C05364=1015.142,141.527,-123.022,166.759,55.577,160.204
C05365=1015.138,141.277,-123.003,166.756,55.588,160.206
C05366=1015.133,141.029,-122.984,166.753,55.599,160.207
C05367=1015.129,140.779,-122.966,166.749,55.609,160.208
C05368=1015.125,140.530,-122.946,166.746,55.621,160.210
C05369=1015.120,140.281,-122.928,166.743,55.631,160.211
C05370=1015.116,140.031,-122.909,166.739,55.642,160.212
C05371=1015.111,139.782,-122.890,166.736,55.653,160.214
C05372=1015.107,139.533,-122.872,166.733,55.663,160.215
C05373=1015.102,139.284,-122.852,166.729,55.674,160.217
C05374=1015.097,139.003,-122.832,166.726,55.687,160.218
C05375=1015.092,138.722,-122.810,166.723,55.699,160.220
C05376=1015.087,138.442,-122.789,166.719,55.711,160.221
C05377=1015.083,138.162,-122.768,166.716,55.723,160.223
C05378=1015.079,137.912,-122.749,166.713,55.734,160.225
C05379=1015.074,137.663,-122.731,166.709,55.745,160.226
C05380=1015.070,137.413,-122.712,166.706,55.756,160.228
C05381=1015.065,137.164,-122.694,166.703,55.766,160.229
C05382=1015.061,136.915,-122.674,166.699,55.778,160.230
C05383=1015.056,136.666,-122.656,166.696,55.788,160.232
C05384=1015.052,136.416,-122.637,166.694,55.799,160.233
C05385=1015.047,136.167,-122.619,166.690,55.810,160.235
C05386=1015.043,135.918,-122.600,166.687,55.821,160.236
C05387=1015.039,135.669,-122.582,166.685,55.832,160.238
C05388=1015.035,135.419,-122.563,166.680,55.843,160.239
C05389=1015.030,135.170,-122.545,166.677,55.853,160.240
C05390=1015.025,134.921,-122.527,166.674,55.865,160.242
C05391=1015.021,134.671,-122.508,166.671,55.875,160.243
C05392=1015.016,134.422,-122.489,166.669,55.887,160.245
C05393=1015.012,134.173,-122.470,166.665,55.897,160.246
C05394=1015.008,133.924,-122.453,166.662,55.908,160.247
C05395=1015.003,133.675,-122.434,166.659,55.919,160.249
C05396=1014.999,133.425,-122.416,166.655,55.930,160.250
C05397=1014.994,133.176,-122.397,166.652,55.941,160.252
C05398=1014.990,132.926,-122.379,166.650,55.952,160.253
C05399=1014.985,132.677,-122.361,166.647,55.962,160.255
C05400=1014.981,132.429,-122.342,166.643,55.974,160.256
C05401=1014.977,132.179,-122.323,166.640,55.984,160.258
C05402=1014.972,131.930,-122.305,166.637,55.995,160.259
C05403=1014.967,131.680,-122.287,166.633,56.006,160.260
C05404=1014.963,131.431,-122.268,166.631,56.017,160.262
C05405=1014.959,131.182,-122.250,166.628,56.028,160.263
C05406=1014.955,130.932,-122.232,166.625,56.038,160.265
C05407=1014.950,130.683,-122.214,166.622,56.050,160.266
C05408=1014.945,130.433,-122.195,166.619,56.060,160.268
C05409=1014.942,130.185,-122.177,166.616,56.071,160.269
C05410=1014.937,129.935,-122.159,166.613,56.082,160.271
C05411=1014.933,129.686,-122.140,166.609,56.093,160.272
C05412=1014.928,129.436,-122.122,166.607,56.103,160.273
C05413=1014.924,129.187,-122.104,166.604,56.115,160.275
C05414=1014.919,128.937,-122.086,166.600,56.126,160.276
C05415=1014.915,128.688,-122.068,166.597,56.136,160.278
C05416=1014.910,128.439,-122.050,166.595,56.147,160.279
C05417=1014.905,128.189,-122.032,166.591,56.158,160.281
C05418=1014.901,127.940,-122.014,166.589,56.170,160.282
C05419=1014.896,127.692,-121.996,166.586,56.180,160.284
C05420=1014.892,127.442,-121.979,166.582,56.192,160.285
C05421=1014.887,127.192,-121.961,166.579,56.202,160.287
C05422=1014.882,126.943,-121.942,166.577,56.213,160.288
C05423=1014.878,126.694,-121.925,166.573,56.224,160.290
C05424=1014.873,126.445,-121.906,166.570,56.235,160.291
C05425=1014.869,126.195,-121.889,166.568,56.246,160.293
C05426=1014.865,125.946,-121.871,166.564,56.257,160.294
C05427=1014.860,125.697,-121.853,166.561,56.268,160.295
C05428=1014.856,125.447,-121.835,166.559,56.279,160.297
C05429=1014.851,125.197,-121.817,166.555,56.290,160.298
C05430=1014.847,124.949,-121.799,166.553,56.301,160.300
C05431=1014.842,124.699,-121.781,166.550,56.312,160.301
C05432=1014.838,124.449,-121.763,166.547,56.322,160.303
C05433=1014.834,124.201,-121.746,166.543,56.334,160.304
C05434=1014.829,123.951,-121.728,166.541,56.345,160.306
C05435=1014.825,123.701,-121.710,166.538,56.355,160.307
C05436=1014.820,123.453,-121.692,166.535,56.366,160.309
C05437=1014.816,123.203,-121.674,166.532,56.377,160.310
C05438=1014.810,122.923,-121.654,166.529,56.390,160.312
C05439=1014.805,122.643,-121.634,166.525,56.402,160.314
C05440=1014.800,122.361,-121.615,166.522,56.414,160.315
C05441=1014.796,122.081,-121.594,166.518,56.426,160.317
C05442=1014.791,121.832,-121.576,166.516,56.437,160.318
C05443=1014.787,121.583,-121.558,166.513,56.448,160.320
C05444=1014.782,121.333,-121.541,166.510,56.459,160.321
C05445=1014.777,121.084,-121.523,166.506,56.470,160.322
C05446=1014.773,120.834,-121.506,166.504,56.481,160.324
C05447=1014.769,120.585,-121.488,166.501,56.492,160.326
C05448=1014.764,120.336,-121.469,166.499,56.502,160.327
C05449=1014.760,120.086,-121.452,166.496,56.513,160.328
C05450=1014.755,119.837,-121.434,166.492,56.524,160.330
C05451=1014.751,119.588,-121.417,166.490,56.535,160.331
C05452=1014.747,119.338,-121.399,166.487,56.546,160.333
C05453=1014.742,119.089,-121.381,166.484,56.556,160.334
C05454=1014.738,118.840,-121.364,166.481,56.567,160.336
C05455=1014.733,118.591,-121.346,166.478,56.577,160.337
C05456=1014.729,118.341,-121.328,166.476,56.589,160.339
C05457=1014.725,118.092,-121.310,166.472,56.600,160.340
C05458=1014.721,117.843,-121.293,166.470,56.610,160.342
C05459=1014.716,117.593,-121.275,166.467,56.621,160.343
C05460=1014.711,117.344,-121.257,166.464,56.632,160.344
C05461=1014.707,117.095,-121.240,166.461,56.642,160.346
C05462=1014.702,116.845,-121.222,166.458,56.653,160.347
C05463=1014.699,116.596,-121.205,166.456,56.664,160.349
C05464=1014.694,116.347,-121.186,166.453,56.675,160.350
C05465=1014.690,116.097,-121.169,166.451,56.685,160.352
C05466=1014.685,115.848,-121.151,166.447,56.696,160.353
C05467=1014.681,115.599,-121.134,166.444,56.707,160.355
C05468=1014.676,115.349,-121.116,166.441,56.718,160.356
C05469=1014.672,115.099,-121.098,166.439,56.728,160.357
C05470=1014.668,114.851,-121.081,166.436,56.739,160.359
C05471=1014.663,114.601,-121.063,166.433,56.750,160.360
C05472=1014.659,114.352,-121.045,166.430,56.760,160.362
C05473=1014.655,114.102,-121.028,166.428,56.771,160.363
C05474=1014.651,113.854,-121.010,166.425,56.781,160.365
C05475=1014.646,113.604,-120.993,166.422,56.792,160.366
C05476=1014.642,113.354,-120.976,166.419,56.803,160.368
C05477=1014.637,113.105,-120.957,166.417,56.813,160.369
C05478=1014.634,112.856,-120.940,166.414,56.824,160.370
C05479=1014.629,112.606,-120.922,166.411,56.835,160.372
C05480=1014.625,112.357,-120.905,166.408,56.845,160.373
C05481=1014.620,112.108,-120.887,166.406,56.856,160.375
C05482=1014.616,111.858,-120.870,166.403,56.867,160.376
C05483=1014.612,111.608,-120.852,166.401,56.878,160.378
C05484=1014.608,111.359,-120.835,166.398,56.889,160.379
C05485=1014.602,111.110,-120.818,166.395,56.899,160.381
C05486=1014.598,110.861,-120.801,166.393,56.910,160.382
C05487=1014.595,110.612,-120.784,166.389,56.921,160.384
C05488=1014.590,110.362,-120.766,166.386,56.932,160.385
C05489=1014.585,110.113,-120.749,166.384,56.942,160.387
C05490=1014.581,109.863,-120.732,166.381,56.953,160.388
C05491=1014.577,109.614,-120.715,166.378,56.964,160.389
C05492=1014.572,109.364,-120.698,166.375,56.974,160.391
C05493=1014.568,109.115,-120.681,166.373,56.986,160.393
C05494=1014.563,108.866,-120.662,166.371,56.996,160.394
C05495=1014.558,108.617,-120.646,166.368,57.007,160.396
C05496=1014.554,108.367,-120.628,166.365,57.018,160.397
C05497=1014.549,108.118,-120.612,166.363,57.028,160.398
C05498=1014.545,107.869,-120.595,166.360,57.039,160.400
C05499=1014.540,107.619,-120.578,166.356,57.050,160.401
C05500=1014.536,107.370,-120.561,166.354,57.061,160.403
C05501=1014.531,107.120,-120.544,166.351,57.072,160.404
C05502=1014.526,106.840,-120.526,166.348,57.084,160.406
C05503=1014.521,106.559,-120.505,166.345,57.096,160.408
C05504=1014.516,106.279,-120.486,166.343,57.108,160.409
C05505=1014.511,105.999,-120.468,166.340,57.120,160.411
C05506=1014.507,105.750,-120.451,166.337,57.131,160.412
C05507=1014.502,105.500,-120.434,166.334,57.142,160.414
C05508=1014.498,105.251,-120.417,166.332,57.152,160.415
C05509=1014.493,105.001,-120.400,166.329,57.163,160.417
C05510=1014.489,104.751,-120.383,166.326,57.174,160.418
C05511=1014.485,104.503,-120.366,166.324,57.184,160.420
C05512=1014.480,104.253,-120.349,166.321,57.195,160.421
C05513=1014.476,104.004,-120.332,166.318,57.206,160.423
C05514=1014.471,103.754,-120.315,166.316,57.217,160.424
C05515=1014.467,103.505,-120.298,166.313,57.227,160.426
C05516=1014.463,103.255,-120.281,166.311,57.238,160.427
C05517=1014.458,103.006,-120.265,166.308,57.249,160.429
C05518=1014.454,102.756,-120.247,166.305,57.259,160.430
C05519=1014.449,102.508,-120.231,166.303,57.270,160.432
C05520=1014.445,102.258,-120.214,166.300,57.281,160.433
C05521=1014.440,102.009,-120.197,166.298,57.292,160.435
C05522=1014.436,101.759,-120.180,166.295,57.302,160.436
C05523=1014.431,101.510,-120.163,166.292,57.313,160.437
C05524=1014.427,101.260,-120.146,166.290,57.324,160.439
C05525=1014.422,101.011,-120.130,166.287,57.334,160.440
C05526=1014.418,100.761,-120.113,166.284,57.344,160.442
C05527=1014.414,100.512,-120.096,166.281,57.355,160.443
C05528=1014.410,100.263,-120.079,166.279,57.366,160.445
C05529=1014.405,100.013,-120.062,166.276,57.377,160.446
C05530=1014.401,99.764,-120.045,166.274,57.387,160.448
C05531=1014.396,99.515,-120.029,166.272,57.398,160.449
C05532=1014.392,99.265,-120.012,166.269,57.408,160.450
C05533=1014.387,99.016,-119.995,166.266,57.418,160.452
C05534=1014.383,98.767,-119.978,166.264,57.429,160.453
C05535=1014.379,98.517,-119.962,166.261,57.440,160.455
C05536=1014.374,98.267,-119.945,166.259,57.451,160.456
C05537=1014.369,98.018,-119.929,166.256,57.461,160.458
C05538=1014.365,97.768,-119.912,166.254,57.472,160.459
C05539=1014.361,97.519,-119.896,166.251,57.483,160.461
C05540=1014.356,97.270,-119.879,166.249,57.494,160.462
C05541=1014.351,97.020,-119.863,166.246,57.504,160.464
C05542=1014.347,96.771,-119.846,166.243,57.515,160.465
C05543=1014.342,96.521,-119.829,166.241,57.526,160.467
C05544=1014.338,96.272,-119.814,166.238,57.537,160.468
C05545=1014.333,96.023,-119.797,166.235,57.547,160.469
C05546=1014.329,95.774,-119.781,166.233,57.557,160.471
C05547=1014.324,95.523,-119.764,166.230,57.568,160.472
C05548=1014.320,95.274,-119.747,166.228,57.579,160.474
C05549=1014.315,95.025,-119.731,166.226,57.589,160.476
C05550=1014.311,94.776,-119.715,166.224,57.600,160.477
C05551=1014.306,94.526,-119.698,166.221,57.611,160.479
C05552=1014.302,94.276,-119.682,166.218,57.621,160.480
C05553=1014.298,94.027,-119.665,166.216,57.632,160.481
C05554=1014.293,93.778,-119.649,166.213,57.642,160.483
C05555=1014.289,93.529,-119.633,166.211,57.653,160.484
C05556=1014.283,93.279,-119.616,166.208,57.664,160.486
C05557=1014.280,93.029,-119.600,166.205,57.674,160.487
C05558=1014.275,92.780,-119.583,166.204,57.684,160.489
C05559=1014.271,92.531,-119.567,166.201,57.695,160.490
C05560=1014.266,92.282,-119.551,166.199,57.706,160.492
C05561=1014.261,92.032,-119.534,166.195,57.716,160.493
C05562=1014.258,91.782,-119.518,166.193,57.727,160.494
C05563=1014.253,91.533,-119.501,166.191,57.738,160.496
C05564=1014.249,91.284,-119.486,166.189,57.747,160.497
C05565=1014.244,91.035,-119.469,166.186,57.758,160.499
C05566=1014.239,90.755,-119.451,166.183,57.770,160.500
C05567=1014.234,90.474,-119.432,166.180,57.782,160.502
C05568=1014.228,90.194,-119.414,166.177,57.794,160.504
C05569=1014.224,89.914,-119.395,166.175,57.805,160.506
C05570=1014.219,89.664,-119.379,166.172,57.815,160.507
C05571=1014.215,89.415,-119.363,166.170,57.826,160.508
C05572=1014.211,89.165,-119.346,166.167,57.836,160.509
C05573=1014.207,88.916,-119.330,166.165,57.847,160.511
C05574=1014.202,88.667,-119.314,166.163,57.857,160.513
C05575=1014.197,88.417,-119.298,166.160,57.868,160.514
C05576=1014.193,88.168,-119.282,166.158,57.878,160.515
C05577=1014.189,87.918,-119.266,166.155,57.889,160.517
C05578=1014.184,87.668,-119.250,166.153,57.900,160.518
C05579=1014.180,87.420,-119.234,166.151,57.910,160.520
C05580=1014.175,87.170,-119.218,166.148,57.920,160.521
C05581=1014.170,86.921,-119.203,166.146,57.931,160.523
C05582=1014.165,86.670,-119.187,166.143,57.941,160.524
C05583=1014.161,86.421,-119.170,166.140,57.952,160.526
C05584=1014.156,86.172,-119.154,166.138,57.963,160.527
C05585=1014.152,85.922,-119.138,166.137,57.973,160.529
C05586=1014.148,85.673,-119.122,166.134,57.984,160.530
C05587=1014.143,85.424,-119.106,166.131,57.994,160.532
C05588=1014.139,85.174,-119.090,166.128,58.004,160.533
C05589=1014.134,84.925,-119.075,166.126,58.015,160.534
C05590=1014.129,84.676,-119.059,166.124,58.026,160.536
C05591=1014.125,84.426,-119.043,166.121,58.036,160.537
C05592=1014.120,84.176,-119.027,166.119,58.047,160.539
C05593=1014.116,83.927,-119.011,166.117,58.057,160.540
C05594=1014.111,83.678,-118.995,166.115,58.067,160.542
C05595=1014.107,83.428,-118.979,166.112,58.078,160.543
C05596=1014.103,83.178,-118.963,166.109,58.088,160.545
C05597=1014.098,82.929,-118.947,166.107,58.099,160.546
C05598=1014.093,82.680,-118.932,166.105,58.109,160.547
C05599=1014.089,82.431,-118.916,166.103,58.119,160.549
C05600=1014.084,82.181,-118.900,166.100,58.130,160.550
C05601=1014.080,81.931,-118.884,166.098,58.140,160.552
C05602=1014.076,81.682,-118.868,166.095,58.150,160.553
C05603=1014.071,81.432,-118.853,166.093,58.161,160.555
C05604=1014.067,81.183,-118.836,166.090,58.171,160.556
C05605=1014.062,80.934,-118.820,166.089,58.182,160.558
C05606=1014.057,80.685,-118.805,166.086,58.192,160.559
C05607=1014.053,80.435,-118.789,166.084,58.203,160.560
C05608=1014.049,80.185,-118.774,166.082,58.212,160.562
C05609=1014.044,79.936,-118.758,166.079,58.222,160.563
C05610=1014.040,79.686,-118.742,166.077,58.233,160.565
C05611=1014.036,79.437,-118.726,166.074,58.243,160.566
C05612=1014.031,79.188,-118.710,166.072,58.254,160.568
C05613=1014.027,78.938,-118.694,166.070,58.263,160.569
C05614=1014.022,78.689,-118.679,166.067,58.274,160.570
C05615=1014.018,78.439,-118.663,166.065,58.284,160.572
C05616=1014.013,78.190,-118.647,166.063,58.294,160.573
C05617=1014.009,77.940,-118.632,166.060,58.304,160.575
C05618=1014.005,77.691,-118.616,166.059,58.315,160.576
C05619=1014.000,77.442,-118.599,166.056,58.325,160.578
C05620=1013.996,77.192,-118.584,166.054,58.335,160.579
C05621=1013.991,76.942,-118.568,166.051,58.345,160.580
C05622=1013.986,76.693,-118.553,166.049,58.356,160.582
C05623=1013.982,76.444,-118.537,166.047,58.365,160.583
C05624=1013.978,76.194,-118.521,166.044,58.376,160.584
C05625=1013.973,75.945,-118.506,166.043,58.386,160.586
C05626=1013.968,75.695,-118.490,166.040,58.396,160.587
C05627=1013.964,75.446,-118.474,166.037,58.406,160.589
C05628=1013.959,75.196,-118.460,166.036,58.417,160.590
C05629=1013.955,74.946,-118.444,166.033,58.427,160.592
C05630=1013.950,74.666,-118.426,166.031,58.439,160.594
C05631=1013.945,74.387,-118.409,166.028,58.450,160.595
C05632=1013.940,74.106,-118.392,166.025,58.462,160.597
C05633=1013.935,73.827,-118.374,166.023,58.473,160.598
C05634=1013.930,73.577,-118.360,166.020,58.483,160.599
C05635=1013.926,73.328,-118.344,166.019,58.494,160.601
C05636=1013.921,73.078,-118.329,166.016,58.504,160.602
C05637=1013.917,72.829,-118.313,166.014,58.513,160.604
C05638=1013.912,72.580,-118.298,166.011,58.524,160.605
C05639=1013.907,72.330,-118.282,166.010,58.534,160.607
C05640=1013.903,72.080,-118.266,166.007,58.544,160.608
C05641=1013.898,71.831,-118.252,166.004,58.554,160.609
C05642=1013.894,71.581,-118.236,166.003,58.564,160.611
C05643=1013.889,71.332,-118.221,166.000,58.574,160.612
C05644=1013.885,71.082,-118.205,165.998,58.584,160.614
C05645=1013.880,70.834,-118.190,165.996,58.595,160.615
C05646=1013.876,70.583,-118.175,165.994,58.605,160.617
C05647=1013.872,70.334,-118.160,165.991,58.615,160.618
C05648=1013.867,70.085,-118.144,165.989,58.625,160.619
C05649=1013.863,69.835,-118.129,165.986,58.635,160.621
C05650=1013.857,69.586,-118.114,165.985,58.645,160.622
C05651=1013.853,69.335,-118.098,165.982,58.655,160.623
C05652=1013.848,69.086,-118.083,165.981,58.665,160.625
C05653=1013.845,68.837,-118.068,165.978,58.676,160.626
C05654=1013.840,68.588,-118.053,165.976,58.685,160.628
C05655=1013.836,68.338,-118.038,165.974,58.695,160.629
C05656=1013.831,68.088,-118.022,165.971,58.705,160.631
C05657=1013.826,67.839,-118.007,165.970,58.715,160.632
C05658=1013.822,67.589,-117.992,165.967,58.725,160.633
C05659=1013.817,67.340,-117.977,165.965,58.735,160.635
C05660=1013.813,67.091,-117.962,165.962,58.745,160.636
C05661=1013.809,66.841,-117.947,165.960,58.755,160.637
C05662=1013.804,66.592,-117.931,165.958,58.765,160.639
C05663=1013.799,66.342,-117.917,165.956,58.775,160.640
C05664=1013.795,66.092,-117.901,165.953,58.785,160.641
C05665=1013.790,65.843,-117.886,165.951,58.795,160.643
C05666=1013.786,65.593,-117.871,165.950,58.805,160.644
C05667=1013.781,65.344,-117.856,165.947,58.815,160.646
C05668=1013.777,65.094,-117.842,165.945,58.825,160.647
C05669=1013.772,64.845,-117.826,165.942,58.835,160.648
C05670=1013.767,64.595,-117.811,165.940,58.845,160.650
C05671=1013.762,64.345,-117.796,165.939,58.855,160.651
C05672=1013.759,64.097,-117.781,165.936,58.865,160.653
C05673=1013.754,63.847,-117.766,165.934,58.875,160.654
C05674=1013.749,63.597,-117.751,165.931,58.885,160.655
C05675=1013.745,63.347,-117.736,165.930,58.895,160.657
C05676=1013.741,63.099,-117.721,165.928,58.904,160.658
C05677=1013.736,62.849,-117.707,165.925,58.915,160.660
C05678=1013.731,62.599,-117.691,165.924,58.924,160.661
C05679=1013.727,62.349,-117.677,165.922,58.934,160.663
C05680=1013.722,62.099,-117.662,165.919,58.944,160.664
C05681=1013.718,61.851,-117.647,165.917,58.954,160.665
C05682=1013.713,61.601,-117.633,165.915,58.964,160.667
C05683=1013.708,61.351,-117.619,165.913,58.974,160.668
C05684=1013.703,61.102,-117.603,165.910,58.984,160.669
C05685=1013.699,60.853,-117.589,165.908,58.994,160.671
C05686=1013.694,60.603,-117.575,165.906,59.005,160.672
C05687=1013.689,60.353,-117.560,165.904,59.014,160.674
C05688=1013.684,60.104,-117.545,165.902,59.024,160.675
C05689=1013.680,59.854,-117.531,165.899,59.034,160.676
C05690=1013.675,59.605,-117.516,165.897,59.043,160.678
C05691=1013.670,59.355,-117.501,165.894,59.054,160.679
C05692=1013.666,59.105,-117.487,165.893,59.064,160.680
C05693=1013.662,58.856,-117.473,165.891,59.073,160.682
C05694=1013.656,58.576,-117.456,165.888,59.085,160.683
C05695=1013.651,58.296,-117.439,165.886,59.096,160.685
C05696=1013.646,58.016,-117.424,165.884,59.107,160.687
C05697=1013.641,57.737,-117.407,165.882,59.118,160.688
C05698=1013.636,57.487,-117.393,165.878,59.127,160.689
C05699=1013.631,57.238,-117.378,165.877,59.137,160.691
C05700=1013.626,56.988,-117.363,165.875,59.147,160.692
C05701=1013.622,56.739,-117.349,165.873,59.157,160.694
C05702=1013.617,56.489,-117.335,165.870,59.166,160.695
C05703=1013.613,56.239,-117.320,165.868,59.176,160.696
C05704=1013.608,55.990,-117.306,165.867,59.186,160.698
C05705=1013.604,55.741,-117.291,165.865,59.196,160.699
C05706=1013.599,55.491,-117.277,165.862,59.205,160.700
C05707=1013.595,55.241,-117.263,165.860,59.215,160.702
C05708=1013.590,54.992,-117.248,165.859,59.225,160.703
C05709=1013.585,54.742,-117.233,165.856,59.234,160.704
C05710=1013.581,54.493,-117.219,165.854,59.244,160.705
C05711=1013.576,54.243,-117.204,165.851,59.253,160.707
C05712=1013.571,53.993,-117.190,165.850,59.263,160.708
C05713=1013.567,53.744,-117.176,165.848,59.273,160.710
C05714=1013.562,53.495,-117.161,165.846,59.282,160.711
C05715=1013.557,53.245,-117.146,165.843,59.293,160.712
C05716=1013.553,52.996,-117.132,165.841,59.302,160.713
C05717=1013.549,52.746,-117.118,165.839,59.311,160.715
C05718=1013.544,52.497,-117.103,165.837,59.321,160.716
C05719=1013.540,52.247,-117.089,165.835,59.330,160.718
C05720=1013.535,51.997,-117.075,165.833,59.340,160.719
C05721=1013.530,51.748,-117.060,165.832,59.349,160.720
C05722=1013.526,51.499,-117.045,165.829,59.358,160.721
C05723=1013.521,51.249,-117.031,165.827,59.369,160.723
C05724=1013.517,50.999,-117.017,165.824,59.378,160.724
C05725=1013.513,50.749,-117.002,165.822,59.387,160.725
C05726=1013.509,50.500,-116.988,165.821,59.397,160.727
C05727=1013.504,50.250,-116.973,165.818,59.406,160.728
C05728=1013.499,50.000,-116.959,165.817,59.416,160.729
C05729=1013.495,49.751,-116.945,165.814,59.425,160.731
C05730=1013.490,49.502,-116.929,165.812,59.434,160.732
C05731=1013.486,49.253,-116.915,165.811,59.444,160.733
C05732=1013.481,49.003,-116.901,165.808,59.453,160.734
C05733=1013.477,48.754,-116.887,165.806,59.462,160.736
C05734=1013.472,48.504,-116.872,165.804,59.471,160.737
C05735=1013.468,48.254,-116.858,165.802,59.481,160.738
C05736=1013.463,48.005,-116.844,165.800,59.490,160.740
C05737=1013.459,47.755,-116.829,165.798,59.499,160.741
C05738=1013.455,47.506,-116.815,165.796,59.509,160.742
C05739=1013.450,47.256,-116.801,165.794,59.518,160.743
C05740=1013.446,47.007,-116.787,165.792,59.528,160.745
C05741=1013.441,46.757,-116.772,165.790,59.537,160.746
C05742=1013.436,46.507,-116.758,165.788,59.546,160.747
C05743=1013.432,46.258,-116.744,165.785,59.555,160.748
C05744=1013.427,46.008,-116.729,165.784,59.564,160.750
C05745=1013.423,45.758,-116.715,165.783,59.573,160.751
C05746=1013.418,45.509,-116.701,165.781,59.583,160.752
C05747=1013.414,45.259,-116.687,165.778,59.592,160.754
C05748=1013.410,45.010,-116.672,165.776,59.601,160.755
C05749=1013.405,44.760,-116.658,165.774,59.610,160.756
C05750=1013.401,44.510,-116.644,165.772,59.619,160.757
C05751=1013.397,44.261,-116.629,165.770,59.628,160.758
C05752=1013.392,44.011,-116.615,165.768,59.637,160.760
C05753=1013.388,43.762,-116.601,165.766,59.646,160.761
C05754=1013.383,43.512,-116.586,165.764,59.655,160.762
C05755=1013.379,43.263,-116.572,165.762,59.664,160.763
C05756=1013.374,43.013,-116.558,165.760,59.674,160.765
C05757=1013.370,42.764,-116.544,165.759,59.682,160.766
C05758=1013.365,42.485,-116.527,165.756,59.693,160.767
C05759=1013.360,42.205,-116.512,165.754,59.703,160.769
C05760=1013.355,41.925,-116.496,165.751,59.712,160.770
C05761=1013.350,41.645,-116.481,165.749,59.722,160.771
C05762=1013.345,41.395,-116.466,165.747,59.732,160.772
C05763=1013.340,41.146,-116.453,165.744,59.741,160.774
C05764=1013.335,40.896,-116.438,165.743,59.749,160.775
C05765=1013.332,40.646,-116.425,165.741,59.759,160.776
C05766=1013.327,40.396,-116.410,165.739,59.768,160.777
C05767=1013.322,40.147,-116.397,165.737,59.777,160.779
C05768=1013.318,39.898,-116.383,165.735,59.786,160.780
C05769=1013.313,39.648,-116.369,165.734,59.795,160.781
C05770=1013.308,39.399,-116.356,165.732,59.804,160.782
C05771=1013.304,39.149,-116.341,165.729,59.813,160.784
C05772=1013.300,38.900,-116.327,165.727,59.822,160.785
C05773=1013.295,38.649,-116.313,165.726,59.831,160.786
C05774=1013.290,38.400,-116.300,165.724,59.840,160.788
C05775=1013.286,38.151,-116.285,165.721,59.849,160.788
C05776=1013.282,37.901,-116.272,165.719,59.858,160.790
C05777=1013.277,37.652,-116.258,165.718,59.867,160.791
C05778=1013.272,37.402,-116.244,165.716,59.876,160.792
C05779=1013.268,37.153,-116.230,165.713,59.884,160.793
C05780=1013.263,36.903,-116.217,165.712,59.893,160.795
C05781=1013.259,36.653,-116.203,165.710,59.902,160.796
C05782=1013.255,36.404,-116.189,165.708,59.911,160.797
C05783=1013.250,36.154,-116.175,165.706,59.919,160.798
C05784=1013.245,35.905,-116.161,165.704,59.928,160.799
C05785=1013.241,35.654,-116.148,165.702,59.938,160.801
C05786=1013.236,35.406,-116.134,165.700,59.947,160.802
C05787=1013.231,35.156,-116.121,165.698,59.955,160.803
C05788=1013.227,34.906,-116.107,165.696,59.964,160.804
C05789=1013.222,34.657,-116.094,165.694,59.973,160.805
C05790=1013.217,34.407,-116.080,165.693,59.982,160.807
C05791=1013.213,34.157,-116.067,165.690,59.990,160.808
C05792=1013.209,33.908,-116.053,165.688,59.999,160.809
C05793=1013.203,33.658,-116.040,165.687,60.008,160.810
C05794=1013.199,33.409,-116.025,165.684,60.017,160.811
C05795=1013.195,33.159,-116.013,165.682,60.026,160.812
C05796=1013.189,32.910,-115.999,165.681,60.035,160.814
C05797=1013.185,32.660,-115.985,165.678,60.043,160.815
C05798=1013.181,32.411,-115.972,165.676,60.052,160.816
C05799=1013.176,32.160,-115.958,165.674,60.060,160.817
C05800=1013.172,31.911,-115.945,165.672,60.069,160.818
C05801=1013.167,31.662,-115.931,165.671,60.078,160.820
C05802=1013.162,31.412,-115.918,165.669,60.087,160.821
C05803=1013.158,31.162,-115.904,165.668,60.095,160.822
C05804=1013.154,30.913,-115.891,165.665,60.104,160.823
C05805=1013.148,30.663,-115.877,165.663,60.112,160.824
C05806=1013.144,30.414,-115.864,165.661,60.121,160.825
C05807=1013.140,30.164,-115.851,165.659,60.129,160.826
C05808=1013.135,29.914,-115.837,165.657,60.138,160.828
C05809=1013.130,29.665,-115.824,165.656,60.146,160.829
C05810=1013.126,29.415,-115.810,165.654,60.155,160.830
C05811=1013.121,29.165,-115.797,165.652,60.163,160.831
C05812=1013.117,28.915,-115.783,165.649,60.172,160.832
C05813=1013.112,28.667,-115.770,165.648,60.181,160.833
C05814=1013.107,28.416,-115.757,165.646,60.189,160.834
C05815=1013.103,28.167,-115.743,165.644,60.197,160.835
C05816=1013.098,27.918,-115.730,165.642,60.206,160.837
C05817=1013.095,27.668,-115.717,165.640,60.214,160.838
C05818=1013.089,27.418,-115.703,165.638,60.222,160.839
C05819=1013.085,27.169,-115.689,165.636,60.231,160.840
C05820=1013.081,26.919,-115.677,165.635,60.240,160.841
C05821=1013.076,26.669,-115.663,165.632,60.248,160.842
C05822=1013.071,26.430,-115.650,165.630,60.256,160.843
C05823=1013.067,26.191,-115.638,165.629,60.264,160.844
C05824=1013.063,25.951,-115.625,165.627,60.272,160.845
C05825=1013.058,25.712,-115.612,165.625,60.280,160.847
C05826=1013.054,25.474,-115.600,165.624,60.288,160.848
C05827=1013.049,25.234,-115.587,165.622,60.296,160.849
C05828=1013.045,24.994,-115.575,165.620,60.303,160.850
C05829=1013.041,24.756,-115.562,165.617,60.312,160.850
C05830=1013.036,24.506,-115.549,165.616,60.321,160.852
C05831=1013.031,24.256,-115.536,165.615,60.329,160.853
C05832=1013.026,24.006,-115.523,165.612,60.337,160.854
C05833=1013.022,23.757,-115.510,165.610,60.345,160.855
C05834=1013.018,23.507,-115.497,165.609,60.353,160.856
C05835=1013.014,23.258,-115.484,165.606,60.362,160.857
C05836=1013.008,23.008,-115.470,165.604,60.370,160.858
C05837=1013.003,22.758,-115.457,165.603,60.378,160.859
C05838=1012.999,22.509,-115.444,165.601,60.386,160.860
C05839=1012.995,22.259,-115.431,165.598,60.394,160.861
C05840=1012.990,22.010,-115.418,165.597,60.402,160.862
C05841=1012.985,21.759,-115.405,165.595,60.410,160.864
C05842=1012.981,21.510,-115.392,165.593,60.418,160.865
C05843=1012.976,21.260,-115.380,165.591,60.427,160.866
C05844=1012.972,21.011,-115.365,165.589,60.435,160.867
C05845=1012.967,20.762,-115.353,165.588,60.443,160.868
C05846=1012.962,20.512,-115.340,165.586,60.451,160.869
C05847=1012.958,20.262,-115.327,165.584,60.459,160.870
C05848=1012.953,20.013,-115.314,165.582,60.468,160.871
C05849=1012.949,19.763,-115.301,165.580,60.476,160.872
C05850=1012.945,19.513,-115.288,165.578,60.484,160.873
C05851=1012.940,19.264,-115.275,165.576,60.491,160.874
C05852=1012.935,19.014,-115.262,165.575,60.499,160.875
C05853=1012.930,18.764,-115.249,165.573,60.507,160.876
C05854=1012.926,18.515,-115.236,165.571,60.515,160.877
C05855=1012.921,18.265,-115.224,165.570,60.523,160.878
C05856=1012.917,18.016,-115.211,165.566,60.531,160.879
C05857=1012.912,17.766,-115.198,165.565,60.539,160.880
C05858=1012.908,17.517,-115.185,165.563,60.547,160.881
C05859=1012.903,17.266,-115.171,165.562,60.555,160.882
C05860=1012.899,17.017,-115.159,165.559,60.562,160.883
C05861=1012.894,16.767,-115.146,165.558,60.570,160.884
C05862=1012.889,16.518,-115.133,165.556,60.578,160.885
C05863=1012.885,16.268,-115.120,165.554,60.586,160.886
C05864=1012.880,16.019,-115.108,165.552,60.594,160.887
C05865=1012.876,15.769,-115.095,165.551,60.602,160.888
C05866=1012.872,15.519,-115.083,165.548,60.609,160.889
C05867=1012.867,15.270,-115.070,165.547,60.617,160.890
C05868=1012.862,15.019,-115.057,165.545,60.625,160.891
C05869=1012.857,14.770,-115.044,165.543,60.632,160.892
C05870=1012.853,14.520,-115.031,165.541,60.641,160.893
C05871=1012.848,14.271,-115.018,165.539,60.648,160.894
C05872=1012.844,14.021,-115.006,165.538,60.656,160.895
C05873=1012.839,13.772,-114.993,165.535,60.663,160.896
C05874=1012.835,13.522,-114.981,165.534,60.671,160.897
C05875=1012.830,13.272,-114.968,165.532,60.679,160.898
C05876=1012.826,13.023,-114.955,165.530,60.687,160.899
C05877=1012.821,12.773,-114.942,165.528,60.694,160.900
C05878=1012.809,24.482,-115.964,165.590,60.551,160.891
C05879=1012.813,24.732,-115.977,165.592,60.543,160.889
C05880=1012.818,24.982,-115.990,165.593,60.535,160.888
C05881=1012.823,25.231,-116.003,165.595,60.527,160.887
C05882=1012.827,25.481,-116.016,165.596,60.519,160.886
C05883=1012.832,25.770,-116.031,165.599,60.509,160.885
C05884=1012.838,26.059,-116.047,165.601,60.500,160.884
C05885=1012.843,26.347,-116.061,165.603,60.490,160.883
C05886=1012.848,26.637,-116.077,165.605,60.481,160.881
C05887=1012.853,26.887,-116.090,165.607,60.473,160.880
C05888=1012.858,27.136,-116.103,165.610,60.465,160.879
C05889=1012.862,27.385,-116.117,165.611,60.457,160.878
C05890=1012.867,27.635,-116.130,165.613,60.449,160.877
C05891=1012.871,27.885,-116.143,165.615,60.441,160.876
C05892=1012.875,28.135,-116.156,165.616,60.433,160.875
C05893=1012.879,28.384,-116.170,165.619,60.424,160.874
C05894=1012.885,28.634,-116.183,165.620,60.416,160.873
C05895=1012.888,28.884,-116.197,165.622,60.408,160.872
C05896=1012.893,29.133,-116.210,165.624,60.400,160.870
C05897=1012.898,29.382,-116.223,165.626,60.391,160.870
C05898=1012.902,29.633,-116.237,165.628,60.383,160.868
C05899=1012.907,29.882,-116.250,165.629,60.375,160.867
C05900=1012.911,30.131,-116.264,165.630,60.367,160.866
C05901=1012.916,30.381,-116.276,165.633,60.358,160.865
C05902=1012.920,30.631,-116.291,165.635,60.350,160.864
C05903=1012.925,30.880,-116.304,165.636,60.342,160.863
C05904=1012.929,31.129,-116.318,165.639,60.334,160.862
C05905=1012.934,31.380,-116.331,165.640,60.325,160.860
C05906=1012.939,31.629,-116.344,165.643,60.316,160.859
C05907=1012.943,31.878,-116.358,165.644,60.308,160.858
C05908=1012.947,32.128,-116.371,165.645,60.300,160.857
C05909=1012.952,32.378,-116.385,165.648,60.291,160.856
C05910=1012.957,32.627,-116.398,165.650,60.283,160.855
C05911=1012.961,32.877,-116.411,165.652,60.275,160.854
C05912=1012.966,33.127,-116.425,165.653,60.266,160.852
C05913=1012.970,33.376,-116.438,165.655,60.258,160.851
C05914=1012.975,33.625,-116.452,165.657,60.249,160.850
C05915=1012.980,33.875,-116.465,165.659,60.241,160.849
C05916=1012.984,34.125,-116.478,165.661,60.232,160.848
C05917=1012.989,34.374,-116.492,165.662,60.223,160.847
C05918=1012.992,34.624,-116.505,165.665,60.215,160.846
C05919=1012.998,34.874,-116.519,165.666,60.206,160.844
C05920=1013.002,35.123,-116.533,165.669,60.198,160.843
C05921=1013.007,35.372,-116.546,165.671,60.188,160.842
C05922=1013.011,35.623,-116.560,165.673,60.180,160.841
C05923=1013.016,35.872,-116.573,165.675,60.171,160.840
C05924=1013.020,36.122,-116.587,165.676,60.163,160.839
C05925=1013.025,36.371,-116.600,165.678,60.154,160.837
C05926=1013.029,36.621,-116.614,165.680,60.146,160.836
C05927=1013.034,36.871,-116.628,165.682,60.137,160.835
C05928=1013.038,37.120,-116.641,165.684,60.129,160.834
C05929=1013.043,37.369,-116.655,165.686,60.120,160.833
C05930=1013.047,37.619,-116.670,165.687,60.112,160.832
C05931=1013.052,37.869,-116.682,165.689,60.102,160.830
C05932=1013.057,38.119,-116.697,165.690,60.094,160.829
C05933=1013.060,38.368,-116.710,165.693,60.085,160.828
C05934=1013.065,38.618,-116.724,165.695,60.076,160.827
C05935=1013.070,38.867,-116.738,165.697,60.068,160.826
C05936=1013.074,39.117,-116.752,165.699,60.059,160.824
C05937=1013.078,39.366,-116.766,165.700,60.050,160.823
C05938=1013.083,39.616,-116.780,165.703,60.042,160.822
C05939=1013.087,39.866,-116.793,165.705,60.032,160.821
C05940=1013.092,40.115,-116.807,165.706,60.024,160.819
C05941=1013.096,40.365,-116.822,165.709,60.015,160.819
C05942=1013.101,40.613,-116.835,165.711,60.006,160.817
C05943=1013.105,40.864,-116.849,165.712,59.997,160.816
C05944=1013.110,41.113,-116.863,165.714,59.988,160.815
C05945=1013.115,41.363,-116.877,165.717,59.980,160.814
C05946=1013.119,41.613,-116.890,165.719,59.971,160.813
C05947=1013.124,41.892,-116.906,165.720,59.961,160.811
C05948=1013.129,42.172,-116.922,165.722,59.951,160.809
C05949=1013.134,42.452,-116.938,165.725,59.941,160.808
C05950=1013.139,42.731,-116.954,165.726,59.931,160.807
C05951=1013.144,42.980,-116.968,165.728,59.922,160.806
C05952=1013.147,43.230,-116.981,165.731,59.914,160.805
C05953=1013.152,43.480,-116.996,165.732,59.905,160.803
C05954=1013.156,43.729,-117.010,165.734,59.896,160.802
C05955=1013.161,43.979,-117.024,165.736,59.886,160.801
C05956=1013.165,44.228,-117.038,165.737,59.878,160.799
C05957=1013.170,44.478,-117.053,165.740,59.869,160.798
C05958=1013.174,44.728,-117.067,165.742,59.860,160.797
C05959=1013.178,44.977,-117.081,165.745,59.851,160.796
C05960=1013.183,45.227,-117.096,165.746,59.842,160.795
C05961=1013.187,45.476,-117.110,165.748,59.833,160.793
C05962=1013.192,45.726,-117.124,165.750,59.824,160.792
C05963=1013.196,45.975,-117.138,165.752,59.815,160.791
C05964=1013.201,46.225,-117.153,165.753,59.806,160.789
C05965=1013.205,46.474,-117.167,165.755,59.797,160.788
C05966=1013.210,46.724,-117.181,165.757,59.788,160.787
C05967=1013.214,46.973,-117.195,165.759,59.779,160.786
C05968=1013.218,47.223,-117.210,165.762,59.769,160.785
C05969=1013.223,47.472,-117.224,165.763,59.761,160.783
C05970=1013.227,47.722,-117.238,165.765,59.752,160.782
C05971=1013.231,47.971,-117.252,165.767,59.742,160.781
C05972=1013.236,48.221,-117.267,165.769,59.733,160.780
C05973=1013.240,48.470,-117.281,165.771,59.724,160.778
C05974=1013.245,48.720,-117.295,165.773,59.715,160.777
C05975=1013.249,48.969,-117.310,165.776,59.706,160.776
C05976=1013.254,49.219,-117.324,165.778,59.697,160.775
C05977=1013.259,49.469,-117.338,165.780,59.687,160.774
C05978=1013.263,49.718,-117.353,165.781,59.679,160.772
C05979=1013.268,49.968,-117.367,165.783,59.669,160.771
C05980=1013.272,50.217,-117.381,165.785,59.660,160.769
C05981=1013.276,50.467,-117.396,165.787,59.651,160.768
C05982=1013.281,50.716,-117.410,165.789,59.641,160.767
C05983=1013.285,50.966,-117.424,165.791,59.632,160.766
C05984=1013.289,51.215,-117.438,165.793,59.622,160.764
C05985=1013.294,51.465,-117.453,165.795,59.613,160.763
C05986=1013.298,51.714,-117.467,165.797,59.604,160.762
C05987=1013.303,51.964,-117.481,165.799,59.594,160.760
C05988=1013.308,52.214,-117.496,165.801,59.585,160.759
C05989=1013.312,52.463,-117.510,165.803,59.576,160.758
C05990=1013.317,52.713,-117.524,165.805,59.566,160.756
C05991=1013.321,52.963,-117.538,165.807,59.557,160.755
C05992=1013.326,53.212,-117.553,165.809,59.548,160.754
C05993=1013.330,53.462,-117.567,165.810,59.538,160.752
C05994=1013.335,53.711,-117.582,165.814,59.528,160.751
C05995=1013.339,53.961,-117.597,165.816,59.519,160.750
C05996=1013.343,54.210,-117.611,165.818,59.509,160.749
C05997=1013.348,54.460,-117.626,165.820,59.500,160.747
C05998=1013.352,54.710,-117.640,165.821,59.490,160.746
C05999=1013.356,54.959,-117.654,165.824,59.481,160.745
C06000=1013.361,55.209,-117.669,165.825,59.471,160.743
C06001=1013.365,55.458,-117.683,165.827,59.462,160.742
C06002=1013.370,55.708,-117.698,165.830,59.452,160.741
C06003=1013.375,55.957,-117.712,165.832,59.443,160.739
C06004=1013.379,56.207,-117.726,165.834,59.433,160.738
C06005=1013.384,56.457,-117.741,165.836,59.424,160.737
C06006=1013.388,56.706,-117.755,165.837,59.414,160.735
C06007=1013.393,56.956,-117.769,165.839,59.404,160.734
C06008=1013.398,57.205,-117.784,165.842,59.395,160.733
C06009=1013.402,57.454,-117.799,165.844,59.385,160.731
C06010=1013.407,57.704,-117.813,165.846,59.376,160.730
C06011=1013.412,57.983,-117.830,165.848,59.365,160.728
C06012=1013.417,58.263,-117.845,165.850,59.354,160.727
C06013=1013.422,58.543,-117.861,165.853,59.342,160.725
C06014=1013.428,58.822,-117.878,165.856,59.332,160.724
C06015=1013.432,59.072,-117.892,165.858,59.322,160.722
C06016=1013.437,59.322,-117.907,165.859,59.312,160.721
C06017=1013.441,59.571,-117.921,165.862,59.302,160.720
C06018=1013.446,59.821,-117.935,165.864,59.293,160.718
C06019=1013.451,60.070,-117.950,165.866,59.283,160.717
C06020=1013.455,60.319,-117.964,165.868,59.273,160.716
C06021=1013.460,60.569,-117.979,165.870,59.263,160.714
C06022=1013.464,60.819,-117.994,165.872,59.253,160.713
C06023=1013.469,61.069,-118.009,165.875,59.243,160.712
C06024=1013.473,61.318,-118.023,165.877,59.234,160.710
C06025=1013.478,61.568,-118.038,165.878,59.224,160.709
C06026=1013.483,61.818,-118.052,165.881,59.213,160.707
C06027=1013.487,62.066,-118.067,165.882,59.204,160.706
C06028=1013.492,62.316,-118.081,165.884,59.194,160.704
C06029=1013.496,62.566,-118.096,165.887,59.183,160.703
C06030=1013.502,62.815,-118.111,165.889,59.174,160.702
C06031=1013.505,63.065,-118.126,165.891,59.165,160.700
C06032=1013.510,63.315,-118.140,165.893,59.154,160.699
C06033=1013.515,63.564,-118.155,165.895,59.144,160.698
C06034=1013.519,63.814,-118.170,165.897,59.135,160.696
C06035=1013.523,64.063,-118.185,165.900,59.125,160.695
C06036=1013.528,64.313,-118.200,165.902,59.115,160.694
C06037=1013.532,64.562,-118.216,165.903,59.106,160.692
C06038=1013.537,64.812,-118.230,165.906,59.095,160.691
C06039=1013.541,65.061,-118.245,165.908,59.085,160.689
C06040=1013.545,65.311,-118.260,165.909,59.076,160.688
C06041=1013.550,65.560,-118.275,165.912,59.065,160.686
C06042=1013.555,65.810,-118.289,165.914,59.056,160.685
C06043=1013.559,66.059,-118.305,165.917,59.046,160.684
C06044=1013.564,66.309,-118.319,165.919,59.036,160.683
C06045=1013.568,66.558,-118.335,165.921,59.026,160.681
C06046=1013.573,66.808,-118.350,165.923,59.016,160.680
C06047=1013.578,67.057,-118.365,165.925,59.006,160.678
C06048=1013.581,67.306,-118.380,165.928,58.996,160.677
C06049=1013.586,67.556,-118.395,165.929,58.986,160.675
C06050=1013.590,67.806,-118.410,165.931,58.977,160.674
C06051=1013.595,68.056,-118.425,165.934,58.966,160.673
C06052=1013.599,68.305,-118.441,165.936,58.956,160.671
C06053=1013.604,68.554,-118.455,165.938,58.946,160.670
C06054=1013.608,68.804,-118.470,165.940,58.936,160.668
C06055=1013.613,69.053,-118.486,165.942,58.927,160.667
C06056=1013.617,69.303,-118.501,165.945,58.916,160.666
C06057=1013.622,69.553,-118.516,165.946,58.907,160.664
C06058=1013.626,69.802,-118.531,165.949,58.896,160.663
C06059=1013.631,70.051,-118.546,165.951,58.887,160.661
C06060=1013.635,70.301,-118.561,165.954,58.876,160.660
C06061=1013.640,70.550,-118.577,165.955,58.867,160.659
C06062=1013.644,70.800,-118.592,165.958,58.856,160.657
C06063=1013.648,71.049,-118.608,165.960,58.847,160.656
C06064=1013.653,71.299,-118.622,165.963,58.836,160.655
C06065=1013.657,71.548,-118.638,165.964,58.827,160.653
C06066=1013.662,71.798,-118.653,165.967,58.816,160.652
C06067=1013.666,72.047,-118.669,165.968,58.806,160.650
C06068=1013.670,72.297,-118.684,165.971,58.796,160.649
C06069=1013.675,72.547,-118.699,165.973,58.786,160.647
C06070=1013.680,72.796,-118.715,165.976,58.776,160.646
C06071=1013.684,73.045,-118.730,165.977,58.766,160.645
C06072=1013.688,73.294,-118.746,165.980,58.756,160.643
C06073=1013.693,73.544,-118.760,165.981,58.745,160.641
C06074=1013.697,73.794,-118.776,165.984,58.735,160.640
C06075=1013.702,74.073,-118.793,165.986,58.724,160.639
C06076=1013.707,74.353,-118.811,165.989,58.713,160.637
C06077=1013.712,74.633,-118.828,165.991,58.701,160.635
C06078=1013.718,74.913,-118.844,165.994,58.690,160.634
C06079=1013.722,75.163,-118.860,165.995,58.679,160.632
C06080=1013.726,75.412,-118.876,165.998,58.669,160.631
C06081=1013.731,75.661,-118.891,166.001,58.659,160.630
C06082=1013.735,75.910,-118.906,166.003,58.649,160.628
C06083=1013.739,76.160,-118.922,166.005,58.638,160.627
C06084=1013.745,76.409,-118.937,166.007,58.628,160.625
C06085=1013.749,76.659,-118.953,166.010,58.618,160.624
C06086=1013.753,76.909,-118.968,166.013,58.608,160.623
C06087=1013.757,77.158,-118.984,166.014,58.597,160.621
C06088=1013.762,77.408,-118.999,166.017,58.587,160.620
C06089=1013.767,77.657,-119.016,166.018,58.577,160.618
C06090=1013.771,77.906,-119.031,166.021,58.567,160.617
C06091=1013.775,78.156,-119.047,166.022,58.557,160.615
C06092=1013.780,78.405,-119.063,166.025,58.547,160.614
C06093=1013.784,78.655,-119.079,166.028,58.536,160.613
C06094=1013.788,78.905,-119.094,166.030,58.527,160.611
C06095=1013.792,79.153,-119.110,166.032,58.516,160.610
C06096=1013.797,79.403,-119.125,166.034,58.506,160.608
C06097=1013.801,79.652,-119.141,166.037,58.496,160.607
C06098=1013.806,79.902,-119.157,166.039,58.485,160.605
C06099=1013.810,80.151,-119.172,166.041,58.475,160.604
C06100=1013.814,80.401,-119.188,166.044,58.465,160.603
C06101=1013.819,80.651,-119.204,166.046,58.454,160.601
C06102=1013.823,80.900,-119.220,166.048,58.444,160.600
C06103=1013.827,81.150,-119.235,166.050,58.434,160.598
C06104=1013.832,81.399,-119.252,166.053,58.423,160.597
C06105=1013.837,81.648,-119.267,166.055,58.414,160.595
C06106=1013.841,81.898,-119.283,166.057,58.403,160.594
C06107=1013.845,82.147,-119.299,166.060,58.393,160.592
C06108=1013.850,82.397,-119.314,166.061,58.382,160.591
C06109=1013.854,82.646,-119.330,166.064,58.372,160.589
C06110=1013.858,82.896,-119.346,166.067,58.361,160.588
C06111=1013.863,83.145,-119.362,166.070,58.351,160.587
C06112=1013.867,83.394,-119.378,166.071,58.341,160.585
C06113=1013.872,83.644,-119.393,166.074,58.330,160.584
C06114=1013.877,83.893,-119.409,166.076,58.320,160.582
C06115=1013.881,84.143,-119.425,166.079,58.309,160.581
C06116=1013.885,84.392,-119.441,166.080,58.299,160.579
C06117=1013.890,84.642,-119.456,166.083,58.289,160.578
C06118=1013.894,84.892,-119.472,166.085,58.278,160.576
C06119=1013.898,85.141,-119.489,166.088,58.267,160.575
C06120=1013.903,85.390,-119.504,166.090,58.257,160.573
C06121=1013.908,85.639,-119.520,166.092,58.246,160.572
C06122=1013.912,85.889,-119.535,166.095,58.236,160.571
C06123=1013.916,86.139,-119.551,166.097,58.225,160.569
C06124=1013.922,86.388,-119.568,166.100,58.215,160.567
C06125=1013.926,86.638,-119.584,166.102,58.204,160.566
C06126=1013.930,86.887,-119.600,166.104,58.194,160.564
C06127=1013.935,87.137,-119.615,166.106,58.183,160.563
C06128=1013.939,87.386,-119.632,166.109,58.173,160.562
C06129=1013.943,87.635,-119.648,166.111,58.162,160.560
C06130=1013.949,87.885,-119.663,166.114,58.151,160.559
C06131=1013.953,88.134,-119.679,166.117,58.141,160.557
C06132=1013.957,88.384,-119.694,166.119,58.130,160.556
C06133=1013.962,88.633,-119.711,166.120,58.120,160.554
C06134=1013.966,88.882,-119.727,166.123,58.110,160.553
C06135=1013.970,89.132,-119.744,166.126,58.099,160.551
C06136=1013.975,89.382,-119.760,166.128,58.088,160.550
C06137=1013.979,89.632,-119.776,166.131,58.078,160.549
C06138=1013.984,89.880,-119.792,166.132,58.068,160.547
C06139=1013.988,90.161,-119.811,166.135,58.056,160.545
C06140=1013.994,90.440,-119.829,166.139,58.044,160.544
C06141=1013.998,90.720,-119.846,166.142,58.032,160.542
C06142=1014.002,91.000,-119.865,166.143,58.021,160.540
C06143=1014.008,91.250,-119.882,166.146,58.010,160.539
C06144=1014.012,91.500,-119.897,166.148,57.999,160.537
C06145=1014.017,91.749,-119.914,166.151,57.989,160.536
C06146=1014.020,91.999,-119.930,166.154,57.978,160.535
C06147=1014.025,92.247,-119.947,166.156,57.967,160.533
C06148=1014.029,92.497,-119.962,166.159,57.957,160.532
C06149=1014.034,92.746,-119.979,166.160,57.947,160.530
C06150=1014.038,92.996,-119.995,166.163,57.936,160.529
C06151=1014.042,93.246,-120.012,166.165,57.925,160.527
C06152=1014.047,93.495,-120.028,166.168,57.915,160.526
C06153=1014.051,93.744,-120.044,166.171,57.904,160.524
C06154=1014.056,93.994,-120.060,166.173,57.894,160.523
C06155=1014.060,94.243,-120.077,166.175,57.883,160.521
C06156=1014.064,94.493,-120.093,166.178,57.872,160.520
C06157=1014.069,94.742,-120.110,166.181,57.862,160.518
C06158=1014.074,94.991,-120.126,166.183,57.851,160.517
C06159=1014.078,95.241,-120.142,166.186,57.840,160.515
C06160=1014.083,95.490,-120.159,166.187,57.830,160.514
C06161=1014.086,95.740,-120.175,166.190,57.819,160.512
C06162=1014.091,95.989,-120.192,166.192,57.808,160.511
C06163=1014.096,96.239,-120.208,166.195,57.797,160.509
C06164=1014.100,96.488,-120.224,166.198,57.787,160.508
C06165=1014.105,96.737,-120.241,166.200,57.777,160.506
C06166=1014.109,96.987,-120.257,166.203,57.766,160.505
C06167=1014.114,97.236,-120.274,166.205,57.755,160.503
C06168=1014.118,97.486,-120.290,166.207,57.744,160.502
C06169=1014.123,97.735,-120.306,166.210,57.733,160.500
C06170=1014.127,97.984,-120.323,166.212,57.723,160.499
C06171=1014.131,98.234,-120.339,166.215,57.712,160.497
C06172=1014.136,98.483,-120.356,166.217,57.701,160.496
C06173=1014.141,98.732,-120.372,166.220,57.690,160.494
C06174=1014.144,98.982,-120.389,166.222,57.679,160.493
C06175=1014.149,99.231,-120.405,166.225,57.669,160.491
C06176=1014.153,99.481,-120.422,166.228,57.659,160.490
C06177=1014.158,99.730,-120.439,166.230,57.648,160.489
C06178=1014.161,99.980,-120.455,166.233,57.637,160.487
C06179=1014.166,100.229,-120.472,166.235,57.626,160.486
C06180=1014.171,100.479,-120.489,166.238,57.616,160.484
C06181=1014.175,100.728,-120.506,166.240,57.605,160.483
C06182=1014.179,100.977,-120.523,166.243,57.594,160.481
C06183=1014.184,101.226,-120.539,166.245,57.583,160.480
C06184=1014.188,101.476,-120.557,166.249,57.573,160.478
C06185=1014.192,101.726,-120.573,166.251,57.562,160.477
C06186=1014.196,101.975,-120.590,166.254,57.552,160.475
C06187=1014.202,102.225,-120.606,166.256,57.541,160.474
C06188=1014.205,102.474,-120.624,166.259,57.530,160.472
C06189=1014.210,102.723,-120.640,166.261,57.519,160.471
C06190=1014.214,102.972,-120.657,166.264,57.509,160.469
C06191=1014.219,103.222,-120.674,166.266,57.498,160.468
C06192=1014.223,103.471,-120.691,166.269,57.487,160.466
C06193=1014.227,103.721,-120.707,166.271,57.476,160.465
C06194=1014.232,103.971,-120.724,166.274,57.466,160.463
C06195=1014.236,104.219,-120.741,166.276,57.455,160.462
C06196=1014.240,104.469,-120.758,166.279,57.444,160.461
C06197=1014.245,104.718,-120.775,166.282,57.433,160.459
C06198=1014.249,104.968,-120.792,166.284,57.423,160.458
C06199=1014.254,105.217,-120.808,166.288,57.412,160.456
C06200=1014.258,105.467,-120.826,166.290,57.401,160.455
C06201=1014.263,105.716,-120.842,166.293,57.390,160.453
C06202=1014.267,105.965,-120.859,166.295,57.379,160.451
C06203=1014.272,106.246,-120.878,166.298,57.367,160.450
C06204=1014.277,106.526,-120.897,166.301,57.355,160.448
C06205=1014.283,106.806,-120.916,166.303,57.342,160.446
C06206=1014.287,107.086,-120.935,166.306,57.330,160.445
C06207=1014.291,107.335,-120.952,166.309,57.320,160.443
C06208=1014.296,107.585,-120.969,166.313,57.309,160.442
C06209=1014.300,107.834,-120.986,166.315,57.298,160.441
C06210=1014.304,108.083,-121.003,166.317,57.286,160.439
C06211=1014.309,108.333,-121.020,166.320,57.276,160.437
C06212=1014.313,108.582,-121.037,166.323,57.265,160.436
C06213=1014.318,108.832,-121.054,166.325,57.254,160.434
C06214=1014.322,109.081,-121.071,166.329,57.243,160.433
C06215=1014.327,109.330,-121.087,166.331,57.232,160.432
C06216=1014.331,109.580,-121.105,166.334,57.222,160.430
C06217=1014.335,109.830,-121.122,166.336,57.210,160.428
C06218=1014.340,110.079,-121.139,166.339,57.200,160.427
C06219=1014.344,110.328,-121.156,166.341,57.189,160.425
C06220=1014.349,110.577,-121.174,166.344,57.178,160.424
C06221=1014.353,110.827,-121.191,166.348,57.167,160.423
C06222=1014.358,111.076,-121.208,166.350,57.156,160.421
C06223=1014.362,111.326,-121.225,166.353,57.146,160.420
C06224=1014.366,111.575,-121.242,166.355,57.134,160.418
C06225=1014.371,111.824,-121.259,166.358,57.124,160.416
C06226=1014.375,112.074,-121.277,166.360,57.113,160.415
C06227=1014.379,112.323,-121.294,166.363,57.102,160.413
C06228=1014.384,112.573,-121.311,166.366,57.091,160.412
C06229=1014.388,112.821,-121.329,166.368,57.081,160.411
C06230=1014.392,113.071,-121.347,166.372,57.070,160.409
C06231=1014.397,113.320,-121.364,166.375,57.059,160.408
C06232=1014.401,113.570,-121.382,166.377,57.048,160.406
C06233=1014.405,113.819,-121.399,166.380,57.038,160.405
C06234=1014.409,114.068,-121.417,166.383,57.027,160.403
C06235=1014.414,114.318,-121.434,166.385,57.016,160.402
C06236=1014.417,114.567,-121.451,166.388,57.006,160.400
C06237=1014.422,114.817,-121.469,166.390,56.994,160.399
C06238=1014.425,115.066,-121.487,166.393,56.984,160.397
C06239=1014.430,115.315,-121.505,166.396,56.972,160.396
C06240=1014.434,115.565,-121.522,166.399,56.962,160.395
C06241=1014.439,115.814,-121.540,166.402,56.951,160.393
C06242=1014.443,116.063,-121.558,166.404,56.940,160.392
C06243=1014.447,116.313,-121.575,166.407,56.930,160.390
C06244=1014.451,116.562,-121.593,166.409,56.918,160.388
C06245=1014.456,116.812,-121.610,166.412,56.908,160.387
C06246=1014.460,117.061,-121.628,166.416,56.897,160.386
C06247=1014.464,117.311,-121.645,166.418,56.886,160.384
C06248=1014.469,117.559,-121.663,166.421,56.875,160.383
C06249=1014.473,117.809,-121.681,166.423,56.864,160.381
C06250=1014.477,118.058,-121.699,166.426,56.853,160.380
C06251=1014.482,118.308,-121.716,166.430,56.842,160.378
C06252=1014.486,118.556,-121.734,166.433,56.832,160.377
C06253=1014.490,118.806,-121.751,166.435,56.821,160.375
C06254=1014.495,119.055,-121.769,166.437,56.810,160.374
C06255=1014.499,119.305,-121.786,166.441,56.799,160.372
C06256=1014.503,119.554,-121.804,166.444,56.788,160.371
C06257=1014.508,119.804,-121.822,166.446,56.777,160.369
C06258=1014.512,120.053,-121.840,166.449,56.766,160.368
C06259=1014.516,120.302,-121.857,166.452,56.755,160.366
C06260=1014.521,120.552,-121.875,166.455,56.744,160.365
C06261=1014.525,120.801,-121.892,166.458,56.733,160.363
C06262=1014.530,121.050,-121.910,166.460,56.722,160.362
C06263=1014.534,121.300,-121.927,166.464,56.711,160.361
C06264=1014.538,121.549,-121.946,166.466,56.700,160.359
C06265=1014.543,121.799,-121.963,166.469,56.689,160.357
C06266=1014.547,122.048,-121.981,166.472,56.679,160.356
C06267=1014.552,122.328,-122.001,166.476,56.666,160.354
C06268=1014.558,122.608,-122.021,166.478,56.653,160.353
C06269=1014.562,122.889,-122.041,166.482,56.642,160.351
C06270=1014.566,123.169,-122.060,166.485,56.629,160.349
C06271=1014.571,123.418,-122.078,166.488,56.618,160.348
C06272=1014.576,123.668,-122.097,166.491,56.606,160.346
C06273=1014.580,123.917,-122.114,166.494,56.596,160.345
C06274=1014.585,124.166,-122.132,166.497,56.585,160.343
C06275=1014.589,124.416,-122.150,166.500,56.573,160.342
C06276=1014.593,124.665,-122.167,166.503,56.563,160.341
C06277=1014.598,124.914,-122.185,166.505,56.551,160.339
C06278=1014.603,125.164,-122.203,166.509,56.540,160.338
C06279=1014.607,125.413,-122.220,166.511,56.529,160.336
C06280=1014.612,125.662,-122.239,166.514,56.519,160.334
C06281=1014.615,125.912,-122.256,166.517,56.507,160.333
C06282=1014.620,126.161,-122.274,166.520,56.496,160.331
C06283=1014.625,126.410,-122.292,166.524,56.485,160.330
C06284=1014.629,126.660,-122.309,166.526,56.474,160.328
C06285=1014.634,126.909,-122.327,166.529,56.463,160.327
C06286=1014.638,127.158,-122.345,166.532,56.452,160.325
C06287=1014.643,127.407,-122.363,166.535,56.441,160.324
C06288=1014.647,127.657,-122.381,166.539,56.429,160.323
C06289=1014.652,127.906,-122.399,166.541,56.419,160.321
C06290=1014.657,128.156,-122.417,166.545,56.407,160.320
C06291=1014.661,128.405,-122.434,166.548,56.396,160.318
C06292=1014.665,128.654,-122.452,166.550,56.385,160.316
C06293=1014.670,128.904,-122.470,166.553,56.373,160.315
C06294=1014.674,129.152,-122.488,166.556,56.363,160.313
C06295=1014.679,129.402,-122.506,166.559,56.351,160.312
C06296=1014.683,129.652,-122.524,166.562,56.341,160.311
C06297=1014.688,129.901,-122.542,166.566,56.330,160.309
C06298=1014.691,130.150,-122.561,166.569,56.318,160.308
C06299=1014.696,130.400,-122.579,166.571,56.308,160.306
C06300=1014.701,130.649,-122.597,166.575,56.297,160.305
C06301=1014.705,130.899,-122.616,166.578,56.286,160.303
C06302=1014.709,131.147,-122.634,166.580,56.275,160.302
C06303=1014.713,131.397,-122.653,166.584,56.263,160.300
C06304=1014.718,131.646,-122.671,166.587,56.253,160.299
C06305=1014.722,131.896,-122.689,166.590,56.242,160.297
C06306=1014.726,132.145,-122.707,166.593,56.231,160.296
C06307=1014.731,132.394,-122.725,166.596,56.220,160.295
C06308=1014.735,132.643,-122.744,166.599,56.208,160.293
C06309=1014.739,132.893,-122.762,166.602,56.198,160.292
C06310=1014.744,133.142,-122.780,166.604,56.187,160.290
C06311=1014.748,133.391,-122.799,166.608,56.176,160.289
C06312=1014.752,133.641,-122.817,166.611,56.165,160.287
C06313=1014.757,133.890,-122.835,166.615,56.153,160.286
C06314=1014.761,134.140,-122.854,166.618,56.143,160.284
C06315=1014.765,134.388,-122.872,166.621,56.131,160.283
C06316=1014.769,134.638,-122.890,166.624,56.121,160.281
C06317=1014.774,134.887,-122.909,166.626,56.110,160.280
C06318=1014.779,135.137,-122.927,166.630,56.099,160.278
C06319=1014.783,135.386,-122.946,166.633,56.087,160.277
C06320=1014.788,135.634,-122.964,166.637,56.076,160.276
C06321=1014.792,135.884,-122.983,166.639,56.065,160.274
C06322=1014.796,136.133,-123.001,166.643,56.054,160.273
C06323=1014.800,136.383,-123.020,166.645,56.043,160.271
C06324=1014.805,136.632,-123.038,166.648,56.033,160.270
C06325=1014.809,136.881,-123.056,166.652,56.021,160.268
C06326=1014.814,137.130,-123.075,166.655,56.010,160.267
C06327=1014.818,137.380,-123.094,166.658,55.999,160.265
C06328=1014.823,137.629,-123.112,166.661,55.988,160.264
C06329=1014.827,137.879,-123.131,166.665,55.977,160.262
C06330=1014.831,138.128,-123.149,166.668,55.966,160.261
C06331=1014.836,138.408,-123.171,166.671,55.953,160.259
C06332=1014.841,138.688,-123.192,166.675,55.942,160.258
C06333=1014.845,138.969,-123.212,166.679,55.929,160.256
C06334=1014.850,139.249,-123.233,166.682,55.917,160.254
C06335=1014.854,139.498,-123.252,166.686,55.906,160.253
C06336=1014.859,139.747,-123.272,166.688,55.895,160.251
C06337=1014.864,139.997,-123.290,166.691,55.884,160.250
C06338=1014.868,140.246,-123.309,166.695,55.873,160.248
C06339=1014.873,140.495,-123.327,166.698,55.862,160.247
C06340=1014.877,140.745,-123.346,166.701,55.850,160.246
C06341=1014.881,140.994,-123.365,166.704,55.840,160.244
C06342=1014.886,141.243,-123.384,166.708,55.828,160.243
C06343=1014.889,141.492,-123.402,166.711,55.818,160.241
C06344=1014.894,141.741,-123.422,166.714,55.806,160.240
C06345=1014.898,141.991,-123.440,166.717,55.796,160.238
C06346=1014.902,142.240,-123.459,166.721,55.784,160.237
C06347=1014.907,142.489,-123.478,166.724,55.774,160.236
C06348=1014.912,142.739,-123.496,166.727,55.762,160.234
C06349=1014.916,142.988,-123.516,166.730,55.752,160.233
C06350=1014.920,143.237,-123.534,166.734,55.740,160.231
C06351=1014.925,143.487,-123.553,166.737,55.730,160.230
C06352=1014.929,143.736,-123.572,166.740,55.718,160.228
C06353=1014.933,143.985,-123.591,166.743,55.708,160.227
C06354=1014.938,144.234,-123.610,166.747,55.696,160.225
C06355=1014.942,144.484,-123.628,166.750,55.685,160.224
C06356=1014.947,144.733,-123.648,166.753,55.674,160.222
C06357=1014.951,144.982,-123.666,166.757,55.663,160.221
C06358=1014.956,145.231,-123.686,166.760,55.652,160.220
C06359=1014.960,145.481,-123.704,166.764,55.641,160.218
C06360=1014.964,145.730,-123.724,166.767,55.630,160.217
C06361=1014.968,145.980,-123.743,166.770,55.619,160.215
C06362=1014.973,146.228,-123.761,166.773,55.608,160.214
C06363=1014.978,146.477,-123.781,166.777,55.597,160.212
C06364=1014.982,146.727,-123.800,166.780,55.586,160.211
C06365=1014.986,146.976,-123.819,166.783,55.575,160.209
C06366=1014.990,147.225,-123.839,166.786,55.564,160.208
C06367=1014.994,147.475,-123.857,166.790,55.553,160.207
C06368=1014.999,147.724,-123.877,166.793,55.542,160.205
C06369=1015.004,147.973,-123.896,166.797,55.531,160.204
C06370=1015.008,148.222,-123.914,166.801,55.520,160.203
C06371=1015.012,148.471,-123.934,166.803,55.509,160.201
C06372=1015.017,148.720,-123.953,166.807,55.498,160.200
C06373=1015.021,148.970,-123.972,166.810,55.487,160.198
C06374=1015.025,149.219,-123.992,166.814,55.476,160.197
C06375=1015.029,149.468,-124.011,166.817,55.465,160.195
C06376=1015.034,149.717,-124.031,166.821,55.454,160.194
C06377=1015.038,149.967,-124.049,166.823,55.443,160.192
C06378=1015.042,150.216,-124.069,166.827,55.432,160.191
C06379=1015.046,150.465,-124.088,166.831,55.421,160.190
C06380=1015.051,150.714,-124.108,166.834,55.410,160.188
C06381=1015.055,150.964,-124.127,166.838,55.399,160.187
C06382=1015.059,151.213,-124.146,166.841,55.388,160.185
C06383=1015.064,151.462,-124.165,166.844,55.377,160.184
C06384=1015.068,151.711,-124.185,166.849,55.366,160.183
C06385=1015.074,151.960,-124.204,166.851,55.355,160.181
C06386=1015.078,152.210,-124.223,166.855,55.343,160.180
C06387=1015.082,152.459,-124.242,166.858,55.333,160.178
C06388=1015.086,152.708,-124.262,166.862,55.321,160.177
C06389=1015.091,152.957,-124.281,166.866,55.311,160.176
C06390=1015.094,153.206,-124.301,166.868,55.300,160.174
C06391=1015.099,153.455,-124.321,166.873,55.289,160.173
C06392=1015.104,153.705,-124.341,166.875,55.278,160.171
C06393=1015.108,153.954,-124.360,166.879,55.267,160.170
C06394=1015.112,154.203,-124.380,166.882,55.256,160.168
C06395=1015.117,154.483,-124.401,166.886,55.243,160.167
C06396=1015.122,154.764,-124.423,166.891,55.231,160.165
C06397=1015.127,155.044,-124.445,166.895,55.219,160.164
C06398=1015.132,155.325,-124.467,166.898,55.207,160.162
C06399=1015.136,155.574,-124.487,166.902,55.195,160.161
C06400=1015.140,155.823,-124.506,166.905,55.185,160.159
C06401=1015.145,156.072,-124.526,166.909,55.173,160.158
C06402=1015.150,156.321,-124.546,166.913,55.162,160.156
C06403=1015.154,156.571,-124.565,166.915,55.151,160.155
C06404=1015.158,156.820,-124.585,166.920,55.141,160.154
C06405=1015.162,157.069,-124.605,166.923,55.129,160.152
C06406=1015.166,157.318,-124.624,166.927,55.119,160.151
C06407=1015.171,157.568,-124.644,166.930,55.107,160.149
C06408=1015.176,157.817,-124.663,166.934,55.096,160.148
C06409=1015.180,158.066,-124.683,166.937,55.086,160.147
C06410=1015.184,158.315,-124.702,166.941,55.074,160.145
C06411=1015.189,158.564,-124.724,166.945,55.063,160.144
C06412=1015.193,158.813,-124.743,166.948,55.053,160.142
C06413=1015.197,159.063,-124.763,166.952,55.042,160.141
C06414=1015.201,159.313,-124.784,166.955,55.031,160.140
C06415=1015.206,159.561,-124.804,166.959,55.021,160.138
C06416=1015.209,159.810,-124.824,166.962,55.010,160.137
C06417=1015.214,160.060,-124.843,166.966,54.999,160.136
C06418=1015.217,160.308,-124.864,166.970,54.989,160.134
C06419=1015.222,160.558,-124.884,166.973,54.977,160.133
C06420=1015.226,160.807,-124.905,166.976,54.967,160.131
C06421=1015.230,161.056,-124.925,166.981,54.956,160.130
C06422=1015.234,161.305,-124.944,166.984,54.945,160.129
C06423=1015.239,161.555,-124.965,166.988,54.934,160.127
C06424=1015.243,161.804,-124.985,166.991,54.923,160.126
C06425=1015.247,162.052,-125.006,166.995,54.913,160.125
C06426=1015.251,162.301,-125.025,166.999,54.902,160.123
C06427=1015.256,162.551,-125.045,167.003,54.890,160.122
C06428=1015.260,162.800,-125.066,167.006,54.880,160.121
C06429=1015.264,163.049,-125.086,167.010,54.869,160.119
C06430=1015.268,163.299,-125.107,167.013,54.858,160.118
C06431=1015.273,163.548,-125.126,167.017,54.848,160.117
C06432=1015.277,163.796,-125.147,167.021,54.836,160.115
C06433=1015.280,164.046,-125.167,167.024,54.826,160.114
C06434=1015.286,164.295,-125.188,167.028,54.815,160.113
C06435=1015.289,164.544,-125.208,167.031,54.804,160.111
C06436=1015.294,164.793,-125.228,167.035,54.794,160.110
C06437=1015.298,165.043,-125.248,167.039,54.782,160.108
C06438=1015.303,165.291,-125.269,167.043,54.772,160.107
C06439=1015.306,165.541,-125.289,167.046,54.761,160.106
C06440=1015.311,165.790,-125.310,167.051,54.750,160.104
C06441=1015.315,166.039,-125.329,167.054,54.740,160.103
C06442=1015.319,166.288,-125.350,167.058,54.728,160.102
C06443=1015.324,166.537,-125.371,167.062,54.718,160.100
C06444=1015.328,166.786,-125.391,167.065,54.707,160.099
C06445=1015.332,167.036,-125.412,167.069,54.696,160.098
C06446=1015.337,167.285,-125.431,167.073,54.685,160.096
C06447=1015.341,167.533,-125.452,167.077,54.674,160.095
C06448=1015.346,167.783,-125.472,167.080,54.663,160.093
C06449=1015.350,168.032,-125.493,167.084,54.652,160.092
C06450=1015.355,168.281,-125.513,167.089,54.642,160.091
C06451=1015.358,168.530,-125.533,167.091,54.631,160.089
C06452=1015.362,168.779,-125.554,167.096,54.620,160.088
C06453=1015.368,169.028,-125.575,167.100,54.609,160.087
C06454=1015.371,169.278,-125.595,167.104,54.598,160.085
C06455=1015.376,169.527,-125.615,167.107,54.587,160.084
C06456=1015.380,169.775,-125.636,167.111,54.576,160.083
C06457=1015.385,170.026,-125.657,167.115,54.565,160.081
C06458=1015.389,170.274,-125.677,167.119,54.555,160.080
C06459=1015.394,170.554,-125.700,167.124,54.542,160.079
C06460=1015.399,170.834,-125.722,167.127,54.530,160.077
C06461=1015.404,171.114,-125.746,167.131,54.518,160.075
C06462=1015.409,171.394,-125.769,167.136,54.506,160.074
C06463=1015.413,171.643,-125.790,167.140,54.495,160.073
C06464=1015.418,171.893,-125.810,167.145,54.484,160.071
C06465=1015.422,172.141,-125.830,167.148,54.473,160.070
C06466=1015.427,172.391,-125.851,167.152,54.462,160.069
C06467=1015.431,172.639,-125.872,167.156,54.451,160.067
C06468=1015.435,172.889,-125.892,167.160,54.440,160.066
C06469=1015.440,173.139,-125.913,167.164,54.429,160.064
C06470=1015.444,173.387,-125.933,167.168,54.418,160.063
C06471=1015.450,173.636,-125.954,167.172,54.407,160.062
C06472=1015.453,173.885,-125.975,167.175,54.396,160.060
C06473=1015.458,174.135,-125.995,167.179,54.386,160.059
C06474=1015.462,174.384,-126.015,167.183,54.374,160.058
C06475=1015.467,174.633,-126.037,167.188,54.364,160.056
C06476=1015.471,174.881,-126.057,167.192,54.352,160.055
C06477=1015.476,175.131,-126.078,167.196,54.342,160.054
C06478=1015.480,175.380,-126.099,167.200,54.331,160.052
C06479=1015.485,175.630,-126.119,167.204,54.320,160.051
C06480=1015.490,175.881,-126.140,167.208,54.309,160.050
C06481=1015.494,176.132,-126.161,167.211,54.298,160.048
C06482=1015.499,176.382,-126.181,167.215,54.287,160.047
C06483=1015.503,176.631,-126.203,167.219,54.276,160.046
C06484=1015.508,176.881,-126.222,167.224,54.265,160.044
C06485=1015.512,177.130,-126.243,167.228,54.254,160.043
C06486=1015.516,177.379,-126.264,167.232,54.243,160.042
C06487=1015.521,177.628,-126.285,167.236,54.232,160.040
C06488=1015.526,177.877,-126.306,167.240,54.222,160.039
C06489=1015.531,178.126,-126.326,167.244,54.210,160.038
C06490=1015.535,178.375,-126.347,167.248,54.199,160.036
C06491=1015.539,178.625,-126.368,167.253,54.189,160.035
C06492=1015.545,178.874,-126.389,167.257,54.177,160.034
C06493=1015.548,179.122,-126.410,167.261,54.167,160.032
C06494=1015.554,179.371,-126.430,167.265,54.155,160.031
C06495=1015.558,179.621,-126.451,167.270,54.145,160.030
C06496=1015.562,179.870,-126.472,167.274,54.134,160.028
C06497=1015.567,180.119,-126.493,167.277,54.122,160.027
C06498=1015.572,180.368,-126.514,167.282,54.112,160.026
C06499=1015.576,180.618,-126.535,167.285,54.101,160.024
C06500=1015.581,180.866,-126.555,167.289,54.090,160.023
C06501=1015.586,181.116,-126.576,167.293,54.079,160.022
C06502=1015.591,181.365,-126.597,167.298,54.069,160.020
C06503=1015.595,181.613,-126.618,167.303,54.057,160.019
C06504=1015.600,181.862,-126.639,167.306,54.047,160.018
C06505=1015.603,182.112,-126.661,167.310,54.036,160.016
C06506=1015.608,182.361,-126.682,167.315,54.025,160.015
C06507=1015.613,182.610,-126.704,167.319,54.015,160.014
C06508=1015.617,182.859,-126.725,167.323,54.004,160.013
C06509=1015.621,183.108,-126.747,167.327,53.993,160.011
C06510=1015.625,183.357,-126.769,167.331,53.983,160.010
C06511=1015.629,183.606,-126.789,167.336,53.972,160.009
C06512=1015.634,183.855,-126.811,167.340,53.962,160.008
C06513=1015.638,184.105,-126.833,167.344,53.950,160.006
C06514=1015.643,184.354,-126.855,167.347,53.940,160.005
C06515=1015.647,184.602,-126.876,167.352,53.930,160.004
C06516=1015.651,184.851,-126.897,167.356,53.919,160.002
C06517=1015.655,185.101,-126.919,167.360,53.908,160.001
C06518=1015.660,185.350,-126.941,167.365,53.898,160.000
C06519=1015.664,185.598,-126.962,167.369,53.887,159.999
C06520=1015.668,185.848,-126.984,167.374,53.877,159.998
C06521=1015.673,186.096,-127.006,167.377,53.866,159.996
C06522=1015.677,186.346,-127.027,167.381,53.855,159.995
C06523=1015.682,186.624,-127.052,167.387,53.844,159.993
C06524=1015.687,186.903,-127.075,167.391,53.831,159.992
C06525=1015.692,187.180,-127.100,167.396,53.820,159.991
C06526=1015.696,187.459,-127.124,167.401,53.808,159.989
C06527=1015.701,187.708,-127.145,167.405,53.797,159.988
C06528=1015.706,187.957,-127.167,167.410,53.787,159.987
C06529=1015.710,188.206,-127.190,167.414,53.775,159.985
C06530=1015.714,188.455,-127.211,167.418,53.765,159.984
C06531=1015.719,188.704,-127.233,167.423,53.755,159.983
C06532=1015.723,188.952,-127.254,167.427,53.743,159.982
C06533=1015.727,189.202,-127.276,167.432,53.733,159.980
C06534=1015.732,189.451,-127.298,167.436,53.722,159.979
C06535=1015.737,189.700,-127.320,167.441,53.712,159.978
C06536=1015.741,189.949,-127.341,167.444,53.701,159.976
C06537=1015.745,190.198,-127.363,167.448,53.691,159.975
C06538=1015.750,190.447,-127.385,167.453,53.680,159.974
C06539=1015.755,190.696,-127.407,167.457,53.669,159.973
C06540=1015.759,190.946,-127.429,167.461,53.659,159.971
C06541=1015.764,191.194,-127.451,167.466,53.648,159.970
C06542=1015.768,191.443,-127.472,167.471,53.638,159.969
C06543=1015.773,191.691,-127.494,167.475,53.627,159.968
C06544=1015.776,191.941,-127.516,167.479,53.616,159.966
C06545=1015.781,192.190,-127.538,167.484,53.606,159.965
C06546=1015.786,192.439,-127.560,167.488,53.595,159.964
C06547=1015.790,192.688,-127.582,167.492,53.584,159.963
C06548=1015.795,192.937,-127.603,167.497,53.574,159.962
C06549=1015.799,193.186,-127.625,167.502,53.563,159.960
C06550=1015.804,193.435,-127.647,167.507,53.552,159.959
C06551=1015.808,193.684,-127.669,167.511,53.541,159.958
C06552=1015.813,193.933,-127.691,167.516,53.531,159.957
C06553=1015.818,194.182,-127.713,167.520,53.520,159.955
C06554=1015.822,194.431,-127.736,167.525,53.509,159.954
C06555=1015.827,194.680,-127.757,167.529,53.499,159.953
C06556=1015.831,194.929,-127.779,167.533,53.488,159.952
C06557=1015.836,195.178,-127.800,167.538,53.477,159.950
C06558=1015.840,195.427,-127.823,167.542,53.467,159.949
C06559=1015.845,195.676,-127.845,167.547,53.457,159.948
C06560=1015.850,195.925,-127.867,167.551,53.446,159.947
C06561=1015.854,196.174,-127.889,167.556,53.435,159.945
C06562=1015.860,196.423,-127.911,167.560,53.425,159.944
C06563=1015.864,196.672,-127.933,167.566,53.413,159.943
C06564=1015.869,196.921,-127.955,167.570,53.403,159.942
C06565=1015.873,197.170,-127.977,167.575,53.392,159.941
C06566=1015.878,197.419,-127.999,167.579,53.381,159.939
C06567=1015.883,197.668,-128.021,167.584,53.371,159.938
C06568=1015.887,197.917,-128.044,167.588,53.361,159.937
C06569=1015.892,198.166,-128.066,167.593,53.350,159.936
C06570=1015.897,198.414,-128.087,167.598,53.339,159.934
C06571=1015.901,198.663,-128.109,167.603,53.328,159.933
C06572=1015.906,198.913,-128.132,167.607,53.318,159.932
C06573=1015.911,199.162,-128.154,167.611,53.307,159.931
C06574=1015.915,199.411,-128.176,167.616,53.297,159.929
C06575=1015.919,199.660,-128.200,167.621,53.286,159.928
C06576=1015.924,199.908,-128.221,167.625,53.276,159.927
C06577=1015.928,200.157,-128.244,167.630,53.265,159.926
C06578=1015.932,200.407,-128.266,167.635,53.255,159.925
C06579=1015.938,200.656,-128.289,167.639,53.245,159.923
C06580=1015.942,200.905,-128.312,167.644,53.234,159.922
C06581=1015.946,201.154,-128.334,167.649,53.224,159.921
C06582=1015.951,201.402,-128.357,167.654,53.213,159.920
C06583=1015.956,201.651,-128.379,167.659,53.202,159.919
C06584=1015.960,201.901,-128.402,167.663,53.192,159.917
C06585=1015.965,202.149,-128.425,167.668,53.182,159.916
C06586=1015.969,202.398,-128.447,167.673,53.171,159.915
C06587=1015.988,203.429,-128.541,168.177,53.241,160.035
C06588=1015.994,203.666,-128.564,168.181,53.232,160.034
C06589=1015.999,203.903,-128.587,168.184,53.223,160.033
C06590=1016.004,204.140,-128.610,168.188,53.215,160.032
C06591=1016.010,204.377,-128.634,168.192,53.205,160.030
C06592=1016.015,204.614,-128.656,168.197,53.197,160.030
C06593=1016.021,204.851,-128.680,168.200,53.188,160.028
C06594=1016.025,205.088,-128.703,168.204,53.179,160.027
C06595=1016.032,205.325,-128.726,168.208,53.170,160.026
C06596=1016.037,205.574,-128.750,168.212,53.161,160.025
C06597=1016.042,205.822,-128.775,168.217,53.152,160.024
C06598=1016.048,206.072,-128.799,168.221,53.143,160.023
C06599=1016.054,206.320,-128.823,168.225,53.134,160.022
C06600=1016.059,206.569,-128.848,168.229,53.125,160.021
C06601=1016.065,206.818,-128.872,168.233,53.116,160.020
C06602=1016.070,207.066,-128.897,168.237,53.107,160.019
C06603=1016.076,207.315,-128.921,168.241,53.098,160.017
C06604=1016.082,207.564,-128.946,168.245,53.089,160.016
C06605=1016.087,207.813,-128.970,168.249,53.079,160.015
C06606=1016.092,208.061,-128.995,168.254,53.071,160.014
C06607=1016.098,208.310,-129.020,168.258,53.062,160.013
C06608=1016.104,208.559,-129.044,168.262,53.052,160.012
C06609=1016.110,208.808,-129.069,168.267,53.044,160.011
C06610=1016.115,209.056,-129.093,168.271,53.035,160.010
C06611=1016.121,209.305,-129.118,168.275,53.025,160.009
C06612=1016.126,209.554,-129.143,168.279,53.017,160.008
C06613=1016.131,209.803,-129.168,168.283,53.008,160.007
C06614=1016.137,210.051,-129.193,168.288,52.999,160.006
C06615=1016.143,210.300,-129.217,168.292,52.990,160.005
C06616=1016.149,210.548,-129.242,168.296,52.982,160.004
C06617=1016.153,210.797,-129.267,168.300,52.972,160.003
C06618=1016.159,211.046,-129.292,168.305,52.964,160.002
C06619=1016.165,211.295,-129.317,168.309,52.955,160.001
C06620=1016.170,211.543,-129.341,168.313,52.946,160.000
C06621=1016.176,211.792,-129.367,168.317,52.938,159.999
C06622=1016.181,212.041,-129.391,168.321,52.929,159.997
C06623=1016.187,212.289,-129.417,168.326,52.920,159.996
C06624=1016.192,212.538,-129.441,168.330,52.911,159.995
C06625=1016.198,212.787,-129.467,168.334,52.903,159.994
C06626=1016.203,213.036,-129.491,168.339,52.894,159.994
C06627=1016.209,213.284,-129.516,168.343,52.885,159.992
C06628=1016.215,213.533,-129.541,168.347,52.876,159.991
C06629=1016.220,213.782,-129.567,168.350,52.868,159.990
C06630=1016.225,214.030,-129.591,168.355,52.859,159.989
C06631=1016.232,214.279,-129.616,168.359,52.851,159.988
C06632=1016.237,214.527,-129.641,168.364,52.842,159.987
C06633=1016.242,214.777,-129.666,168.368,52.833,159.986
C06634=1016.248,215.025,-129.691,168.373,52.825,159.985
C06635=1016.254,215.274,-129.716,168.376,52.816,159.984
C06636=1016.260,215.523,-129.741,168.380,52.807,159.983
C06637=1016.265,215.772,-129.766,168.385,52.799,159.982
C06638=1016.271,216.020,-129.792,168.389,52.790,159.981
C06639=1016.276,216.268,-129.817,168.394,52.782,159.980
C06640=1016.282,216.517,-129.841,168.398,52.773,159.980
C06641=1016.288,216.766,-129.867,168.401,52.765,159.978
C06642=1016.293,217.014,-129.892,168.406,52.756,159.977
C06643=1016.299,217.264,-129.917,168.411,52.748,159.976
C06644=1016.305,217.512,-129.942,168.415,52.739,159.976
C06645=1016.310,217.761,-129.968,168.420,52.731,159.975
C06646=1016.316,218.009,-129.993,168.423,52.723,159.974
C06647=1016.322,218.257,-130.018,168.428,52.714,159.973
C06648=1016.327,218.496,-130.042,168.431,52.706,159.972
C06649=1016.332,218.736,-130.067,168.436,52.698,159.971
C06650=1016.338,218.975,-130.091,168.440,52.690,159.970
C06651=1016.343,219.214,-130.116,168.444,52.682,159.969
C06652=1016.348,219.453,-130.140,168.448,52.674,159.968
C06653=1016.354,219.692,-130.164,168.452,52.666,159.967
C06654=1016.359,219.931,-130.189,168.456,52.658,159.966
C06655=1016.365,220.171,-130.213,168.460,52.650,159.965
C06656=1016.370,220.420,-130.239,168.465,52.642,159.965
C06657=1016.376,220.668,-130.264,168.470,52.634,159.964
C06658=1016.381,220.917,-130.290,168.473,52.626,159.963
C06659=1016.387,221.165,-130.315,168.478,52.617,159.962
C06660=1016.392,221.414,-130.341,168.482,52.609,159.961
C06661=1016.398,221.663,-130.367,168.486,52.601,159.960
C06662=1016.404,221.911,-130.392,168.490,52.592,159.959
C06663=1016.409,222.160,-130.418,168.496,52.584,159.958
C06664=1016.415,222.408,-130.443,168.499,52.576,159.957
C06665=1016.420,222.657,-130.469,168.504,52.568,159.956
C06666=1016.427,222.906,-130.494,168.507,52.560,159.955
C06667=1016.432,223.154,-130.520,168.512,52.551,159.954
C06668=1016.438,223.403,-130.545,168.517,52.544,159.954
C06669=1016.443,223.652,-130.571,168.520,52.536,159.952
C06670=1016.449,223.900,-130.598,168.525,52.527,159.952
C06671=1016.455,224.148,-130.623,168.530,52.519,159.951
C06672=1016.460,224.397,-130.649,168.534,52.511,159.950
C06673=1016.466,224.646,-130.674,168.538,52.503,159.949
C06674=1016.472,224.895,-130.700,168.542,52.495,159.948
C06675=1016.478,225.143,-130.725,168.547,52.487,159.947
C06676=1016.483,225.392,-130.751,168.551,52.479,159.946
C06677=1016.489,225.640,-130.776,168.555,52.471,159.945
C06678=1016.495,225.889,-130.803,168.560,52.463,159.945
C06679=1016.500,226.138,-130.829,168.564,52.455,159.944
C06680=1016.506,226.386,-130.854,168.568,52.447,159.943
C06681=1016.511,226.635,-130.880,168.573,52.439,159.942
C06682=1016.517,226.883,-130.906,168.577,52.431,159.941
C06683=1016.523,227.132,-130.932,168.582,52.423,159.940
C06684=1016.529,227.381,-130.958,168.586,52.416,159.939
C06685=1016.535,227.629,-130.984,168.591,52.407,159.938
C06686=1016.540,227.878,-131.010,168.595,52.400,159.938
C06687=1016.545,228.126,-131.036,168.599,52.392,159.937
C06688=1016.551,228.375,-131.062,168.603,52.384,159.936
C06689=1016.556,228.624,-131.088,168.608,52.376,159.935
C06690=1016.562,228.872,-131.114,168.612,52.369,159.934
C06691=1016.568,229.121,-131.140,168.617,52.361,159.934
C06692=1016.574,229.370,-131.166,168.621,52.353,159.933
C06693=1016.579,229.618,-131.193,168.626,52.345,159.932
C06694=1016.585,229.867,-131.219,168.630,52.338,159.931
C06695=1016.590,230.115,-131.245,168.634,52.329,159.930
C06696=1016.596,230.363,-131.271,168.638,52.322,159.929
C06697=1016.602,230.612,-131.297,168.642,52.315,159.928
C06698=1016.607,230.861,-131.323,168.647,52.306,159.928
C06699=1016.613,231.109,-131.350,168.651,52.299,159.927
C06700=1016.619,231.357,-131.376,168.656,52.291,159.926
C06701=1016.624,231.606,-131.402,168.660,52.284,159.925
C06702=1016.630,231.855,-131.429,168.665,52.276,159.925
C06703=1016.636,232.104,-131.455,168.669,52.268,159.924
C06704=1016.641,232.352,-131.482,168.673,52.261,159.923
C06705=1016.647,232.600,-131.508,168.678,52.253,159.922
C06706=1016.653,232.849,-131.534,168.682,52.246,159.921
C06707=1016.658,233.098,-131.561,168.687,52.238,159.921
C06708=1016.663,233.332,-131.585,168.691,52.231,159.920
C06709=1016.669,233.568,-131.610,168.695,52.224,159.919
C06710=1016.675,233.803,-131.635,168.700,52.217,159.918
C06711=1016.680,234.037,-131.660,168.704,52.210,159.918
C06712=1016.685,234.273,-131.685,168.708,52.202,159.917
C06713=1016.690,234.507,-131.710,168.712,52.196,159.916
C06714=1016.696,234.742,-131.736,168.717,52.188,159.915
C06715=1016.702,234.977,-131.761,168.721,52.181,159.915
C06716=1016.707,235.226,-131.786,168.725,52.174,159.914
C06717=1016.713,235.475,-131.813,168.729,52.166,159.913
C06718=1016.719,235.723,-131.840,168.734,52.159,159.912
C06719=1016.725,235.971,-131.866,168.738,52.152,159.911
C06720=1016.731,236.220,-131.893,168.742,52.144,159.911
C06721=1016.735,236.469,-131.920,168.747,52.137,159.910
C06722=1016.741,236.717,-131.946,168.751,52.129,159.909
C06723=1016.747,236.966,-131.973,168.756,52.122,159.908
C06724=1016.753,237.214,-132.000,168.760,52.114,159.908
C06725=1016.758,237.462,-132.026,168.764,52.107,159.907
C06726=1016.764,237.711,-132.053,168.770,52.100,159.906
C06727=1016.770,237.959,-132.079,168.774,52.093,159.906
C06728=1016.776,238.207,-132.106,168.778,52.085,159.905
C06729=1016.782,238.456,-132.133,168.783,52.078,159.904
C06730=1016.788,238.705,-132.160,168.787,52.070,159.903
C06731=1016.794,238.953,-132.186,168.791,52.063,159.902
C06732=1016.799,239.202,-132.213,168.796,52.057,159.902
C06733=1016.804,239.450,-132.240,168.801,52.049,159.901
C06734=1016.810,239.699,-132.267,168.805,52.042,159.900
C06735=1016.816,239.947,-132.294,168.810,52.035,159.900
C06736=1016.821,240.196,-132.321,168.815,52.027,159.899
C06737=1016.827,240.444,-132.347,168.819,52.020,159.898
C06738=1016.833,240.693,-132.375,168.823,52.014,159.898
C06739=1016.838,240.942,-132.402,168.827,52.006,159.897
C06740=1016.844,241.189,-132.429,168.833,51.999,159.896
C06741=1016.850,241.438,-132.456,168.837,51.992,159.896
C06742=1016.855,241.686,-132.483,168.841,51.985,159.895
C06743=1016.861,241.936,-132.510,168.845,51.977,159.894
C06744=1016.867,242.184,-132.537,168.850,51.971,159.893
C06745=1016.873,242.432,-132.563,168.855,51.963,159.893
C06746=1016.878,242.680,-132.591,168.859,51.957,159.892
C06747=1016.884,242.929,-132.618,168.864,51.949,159.891
C06748=1016.890,243.178,-132.646,168.868,51.943,159.891
C06749=1016.896,243.426,-132.673,168.872,51.935,159.890
C06750=1016.901,243.674,-132.700,168.878,51.929,159.889
C06751=1016.907,243.923,-132.727,168.882,51.922,159.889
C06752=1016.912,244.171,-132.755,168.886,51.915,159.888
C06753=1016.918,244.420,-132.782,168.891,51.908,159.887
C06754=1016.924,244.668,-132.810,168.895,51.901,159.887
C06755=1016.929,244.917,-132.837,168.900,51.894,159.886
C06756=1016.934,245.165,-132.865,168.904,51.888,159.885
C06757=1016.941,245.414,-132.892,168.910,51.881,159.885
C06758=1016.946,245.662,-132.920,168.914,51.873,159.884
C06759=1016.952,245.910,-132.947,168.918,51.867,159.884
C06760=1016.958,246.159,-132.975,168.923,51.860,159.883
C06761=1016.963,246.408,-133.002,168.927,51.853,159.882
C06762=1016.969,246.655,-133.029,168.932,51.847,159.882
C06763=1016.974,246.904,-133.057,168.936,51.840,159.881
C06764=1016.980,247.152,-133.084,168.942,51.833,159.881
C06765=1016.985,247.401,-133.112,168.946,51.826,159.880
C06766=1016.991,247.649,-133.140,168.950,51.819,159.879
C06767=1016.997,247.898,-133.167,168.955,51.813,159.879
C06768=1017.002,248.129,-133.193,168.959,51.806,159.878
C06769=1017.008,248.361,-133.219,168.963,51.800,159.877
C06770=1017.013,248.592,-133.245,168.968,51.794,159.877
C06771=1017.019,248.825,-133.270,168.971,51.788,159.876
C06772=1017.023,249.056,-133.296,168.976,51.781,159.876
C06773=1017.029,249.288,-133.322,168.981,51.775,159.875
C06774=1017.034,249.519,-133.348,168.985,51.769,159.875
C06775=1017.040,249.750,-133.373,168.989,51.763,159.874
C06776=1017.045,249.999,-133.401,168.994,51.756,159.873
C06777=1017.051,250.247,-133.428,168.998,51.749,159.873
C06778=1017.057,250.496,-133.456,169.003,51.743,159.872
C06779=1017.063,250.744,-133.483,169.007,51.736,159.872
C06780=1017.069,250.993,-133.511,169.013,51.729,159.871
C06781=1017.074,251.241,-133.539,169.017,51.723,159.870
C06782=1017.080,251.489,-133.567,169.022,51.716,159.870
C06783=1017.086,251.738,-133.594,169.027,51.710,159.869
C06784=1017.091,251.986,-133.622,169.031,51.703,159.869
C06785=1017.098,252.234,-133.650,169.036,51.697,159.868
C06786=1017.103,252.482,-133.678,169.040,51.690,159.868
C06787=1017.110,252.731,-133.706,169.045,51.684,159.867
C06788=1017.115,252.980,-133.733,169.049,51.677,159.866
C06789=1017.121,253.228,-133.761,169.054,51.670,159.866
C06790=1017.127,253.476,-133.789,169.060,51.664,159.865
C06791=1017.133,253.725,-133.817,169.064,51.657,159.865
C06792=1017.138,253.973,-133.845,169.069,51.651,159.864
C06793=1017.145,254.221,-133.873,169.073,51.644,159.863
C06794=1017.151,254.469,-133.901,169.078,51.637,159.863
C06795=1017.157,254.718,-133.928,169.082,51.631,159.862
C06796=1017.163,254.967,-133.956,169.087,51.624,159.862
C06797=1017.168,255.215,-133.984,169.092,51.618,159.861
C06798=1017.175,255.464,-134.012,169.096,51.612,159.861
C06799=1017.180,255.712,-134.040,169.101,51.605,159.860
C06800=1017.186,255.960,-134.068,169.106,51.599,159.860
C06801=1017.193,256.209,-134.096,169.110,51.592,159.859
C06802=1017.198,256.457,-134.124,169.116,51.585,159.858
C06803=1017.204,256.706,-134.152,169.120,51.579,159.858
C06804=1017.210,256.953,-134.179,169.125,51.573,159.857
C06805=1017.216,257.202,-134.208,169.130,51.567,159.857
C06806=1017.223,257.451,-134.235,169.135,51.560,159.856
C06807=1017.228,257.699,-134.263,169.139,51.554,159.856
C06808=1017.234,257.947,-134.292,169.144,51.548,159.855
C06809=1017.241,258.195,-134.320,169.149,51.541,159.855
C06810=1017.246,258.443,-134.348,169.153,51.535,159.854
C06811=1017.252,258.692,-134.376,169.158,51.529,159.854
C06812=1017.259,258.940,-134.404,169.163,51.522,159.853
C06813=1017.264,259.189,-134.432,169.167,51.516,159.853
C06814=1017.270,259.437,-134.460,169.172,51.510,159.852
C06815=1017.277,259.686,-134.488,169.177,51.503,159.852
C06816=1017.283,259.933,-134.517,169.182,51.497,159.851
C06817=1017.289,260.182,-134.545,169.187,51.491,159.851
C06818=1017.295,260.431,-134.573,169.191,51.485,159.850
C06819=1017.300,260.678,-134.602,169.196,51.479,159.850
C06820=1017.306,260.927,-134.630,169.201,51.473,159.849
C06821=1017.312,261.175,-134.659,169.206,51.466,159.849
C06822=1017.318,261.424,-134.688,169.211,51.461,159.848
C06823=1017.324,261.672,-134.716,169.215,51.454,159.848
C06824=1017.329,261.920,-134.745,169.220,51.448,159.847
C06825=1017.335,262.169,-134.774,169.225,51.442,159.847
C06826=1017.341,262.417,-134.803,169.230,51.436,159.846
C06827=1017.347,262.665,-134.831,169.235,51.430,159.846
C06828=1017.353,262.896,-134.857,169.239,51.425,159.845
C06829=1017.358,263.127,-134.884,169.244,51.419,159.845
C06830=1017.363,263.357,-134.911,169.248,51.413,159.845
C06831=1017.369,263.588,-134.937,169.253,51.407,159.844
C06832=1017.375,263.819,-134.964,169.257,51.402,159.844
C06833=1017.381,264.049,-134.990,169.262,51.396,159.843
C06834=1017.386,264.280,-135.017,169.266,51.391,159.843
C06835=1017.391,264.511,-135.044,169.271,51.385,159.843
C06836=1017.398,264.759,-135.073,169.276,51.379,159.842
C06837=1017.403,265.008,-135.101,169.280,51.374,159.842
C06838=1017.409,265.256,-135.130,169.285,51.368,159.841
C06839=1017.415,265.504,-135.159,169.290,51.362,159.841
C06840=1017.421,265.753,-135.188,169.295,51.356,159.840
C06841=1017.427,266.001,-135.217,169.300,51.350,159.840
C06842=1017.432,266.248,-135.246,169.305,51.344,159.839
C06843=1017.439,266.497,-135.275,169.310,51.338,159.839
C06844=1017.445,266.745,-135.303,169.315,51.332,159.839
C06845=1017.451,266.993,-135.332,169.320,51.326,159.838
C06846=1017.456,267.242,-135.362,169.325,51.320,159.838
C06847=1017.463,267.490,-135.391,169.330,51.315,159.837
C06848=1017.469,267.738,-135.420,169.334,51.309,159.837
C06849=1017.475,267.987,-135.448,169.339,51.303,159.837
C06850=1017.480,268.235,-135.478,169.344,51.298,159.836
C06851=1017.486,268.483,-135.507,169.349,51.292,159.836
C06852=1017.492,268.731,-135.536,169.354,51.286,159.835
C06853=1017.499,268.979,-135.565,169.359,51.280,159.835
C06854=1017.504,269.227,-135.594,169.364,51.274,159.835
C06855=1017.510,269.476,-135.623,169.369,51.269,159.834
C06856=1017.517,269.724,-135.653,169.374,51.263,159.834
C06857=1017.522,269.972,-135.682,169.378,51.257,159.833
C06858=1017.528,270.220,-135.711,169.383,51.252,159.833
C06859=1017.534,270.469,-135.741,169.388,51.246,159.833
C06860=1017.540,270.717,-135.770,169.393,51.241,159.832
C06861=1017.546,270.965,-135.799,169.398,51.235,159.832
C06862=1017.552,271.213,-135.829,169.403,51.229,159.832
C06863=1017.558,271.462,-135.858,169.408,51.223,159.831
C06864=1017.564,271.710,-135.887,169.413,51.218,159.831
C06865=1017.570,271.958,-135.917,169.418,51.213,159.831
C06866=1017.576,272.206,-135.946,169.423,51.207,159.830
C06867=1017.582,272.454,-135.976,169.428,51.201,159.830
C06868=1017.588,272.702,-136.005,169.433,51.196,159.830
C06869=1017.594,272.951,-136.034,169.438,51.190,159.829
C06870=1017.600,273.198,-136.064,169.442,51.185,159.829
C06871=1017.606,273.447,-136.094,169.448,51.180,159.829
C06872=1017.612,273.695,-136.123,169.453,51.174,159.828
C06873=1017.617,273.943,-136.152,169.458,51.168,159.828
C06874=1017.624,274.191,-136.182,169.463,51.163,159.828
C06875=1017.630,274.439,-136.212,169.468,51.157,159.827
C06876=1017.636,274.687,-136.241,169.473,51.151,159.827
C06877=1017.641,274.936,-136.270,169.478,51.146,159.827
C06878=1017.648,275.184,-136.301,169.483,51.141,159.826
C06879=1017.654,275.432,-136.330,169.488,51.136,159.826
C06880=1017.661,275.680,-136.360,169.493,51.130,159.826
C06881=1017.666,275.928,-136.390,169.499,51.125,159.825
C06882=1017.672,276.176,-136.419,169.504,51.119,159.825
C06883=1017.678,276.424,-136.449,169.508,51.113,159.824
C06884=1017.684,276.672,-136.478,169.513,51.108,159.824
C06885=1017.690,276.920,-136.508,169.519,51.103,159.824
C06886=1017.696,277.169,-136.538,169.524,51.097,159.824
C06887=1017.702,277.417,-136.569,169.529,51.092,159.824
C06888=1017.708,277.650,-136.597,169.534,51.088,159.823
C06889=1017.713,277.883,-136.625,169.538,51.083,159.823
C06890=1017.719,278.116,-136.653,169.544,51.078,159.823
C06891=1017.725,278.349,-136.681,169.548,51.073,159.823
C06892=1017.730,278.582,-136.709,169.552,51.068,159.822
C06893=1017.736,278.815,-136.737,169.557,51.062,159.822
C06894=1017.741,279.047,-136.766,169.562,51.058,159.822
C06895=1017.747,279.281,-136.794,169.566,51.053,159.821
C06896=1017.754,279.529,-136.823,169.572,51.048,159.821
C06897=1017.759,279.776,-136.854,169.577,51.043,159.821
C06898=1017.766,280.025,-136.884,169.583,51.038,159.821
C06899=1017.771,280.273,-136.914,169.588,51.032,159.820
C06900=1017.778,280.521,-136.944,169.592,51.027,159.820
C06901=1017.784,280.769,-136.974,169.598,51.022,159.820
C06902=1017.790,281.017,-137.005,169.603,51.017,159.820
C06903=1017.796,281.266,-137.034,169.608,51.012,159.820
C06904=1017.802,281.513,-137.064,169.614,51.006,159.819
C06905=1017.808,281.761,-137.095,169.618,51.001,159.819
C06906=1017.814,282.010,-137.125,169.623,50.996,159.819
C06907=1017.820,282.257,-137.156,169.629,50.991,159.818
C06908=1017.826,282.505,-137.186,169.634,50.986,159.818
C06909=1017.833,282.754,-137.215,169.640,50.981,159.818
C06910=1017.839,283.002,-137.246,169.644,50.976,159.818
C06911=1017.845,283.250,-137.276,169.649,50.970,159.817
C06912=1017.851,283.498,-137.307,169.655,50.965,159.817
C06913=1017.858,283.746,-137.337,169.660,50.960,159.817
C06914=1017.864,283.994,-137.367,169.666,50.955,159.817
C06915=1017.870,284.242,-137.398,169.670,50.950,159.817
C06916=1017.876,284.490,-137.428,169.675,50.945,159.816
C06917=1017.883,284.738,-137.458,169.681,50.940,159.816
C06918=1017.889,284.986,-137.488,169.686,50.935,159.816
C06919=1017.895,285.234,-137.519,169.691,50.930,159.816
C06920=1017.901,285.482,-137.549,169.697,50.926,159.816
C06921=1017.907,285.730,-137.580,169.702,50.921,159.816
C06922=1017.913,285.979,-137.611,169.708,50.916,159.815
C06923=1017.919,286.226,-137.642,169.712,50.911,159.815
C06924=1017.926,286.474,-137.672,169.717,50.906,159.815
C06925=1017.931,286.722,-137.703,169.723,50.901,159.815
C06926=1017.938,286.971,-137.733,169.728,50.896,159.814
C06927=1017.944,287.219,-137.764,169.733,50.892,159.814
C06928=1017.950,287.466,-137.795,169.739,50.887,159.814
C06929=1017.956,287.714,-137.826,169.744,50.882,159.814
C06930=1017.963,287.963,-137.856,169.750,50.877,159.814
C06931=1017.969,288.210,-137.887,169.754,50.873,159.814
C06932=1017.975,288.459,-137.918,169.760,50.867,159.814
C06933=1017.981,288.706,-137.948,169.765,50.862,159.813
C06934=1017.987,288.955,-137.980,169.771,50.858,159.813
C06935=1017.993,289.202,-138.011,169.776,50.853,159.813
C06936=1017.999,289.451,-138.041,169.781,50.848,159.813
C06937=1018.005,289.698,-138.073,169.787,50.844,159.813
C06938=1018.012,289.947,-138.103,169.792,50.839,159.813
C06939=1018.018,290.194,-138.134,169.797,50.834,159.812
C06940=1018.024,290.442,-138.165,169.803,50.830,159.812
C06941=1018.031,290.690,-138.196,169.808,50.824,159.812
C06942=1018.037,290.938,-138.227,169.814,50.820,159.812
C06943=1018.044,291.186,-138.258,169.818,50.815,159.812
C06944=1018.049,291.434,-138.289,169.824,50.810,159.812
C06945=1018.055,291.682,-138.321,169.830,50.806,159.812
C06946=1018.062,291.931,-138.351,169.835,50.801,159.812
C06947=1018.068,292.178,-138.382,169.840,50.797,159.812
C06948=1018.074,292.417,-138.412,169.846,50.792,159.812
C06949=1018.080,292.656,-138.443,169.850,50.788,159.811
C06950=1018.085,292.895,-138.473,169.856,50.783,159.811
C06951=1018.091,293.134,-138.503,169.861,50.779,159.811
C06952=1018.098,293.373,-138.533,169.867,50.775,159.811
C06953=1018.104,293.613,-138.563,169.871,50.770,159.811
C06954=1018.109,293.852,-138.594,169.877,50.766,159.811
C06955=1018.115,294.091,-138.624,169.882,50.762,159.811
C06956=1018.121,294.338,-138.655,169.888,50.757,159.811
C06957=1018.127,294.587,-138.687,169.893,50.753,159.811
C06958=1018.134,294.834,-138.719,169.899,50.749,159.811
C06959=1018.139,295.082,-138.751,169.904,50.744,159.811
C06960=1018.145,295.330,-138.783,169.909,50.740,159.810
C06961=1018.152,295.578,-138.814,169.915,50.735,159.811
C06962=1018.158,295.826,-138.846,169.921,50.731,159.811
C06963=1018.164,296.073,-138.877,169.926,50.727,159.810
C06964=1018.170,296.322,-138.909,169.931,50.722,159.810
C06965=1018.177,296.570,-138.941,169.937,50.717,159.810
C06966=1018.182,296.817,-138.972,169.942,50.713,159.810
C06967=1018.189,297.065,-139.004,169.948,50.709,159.810
C06968=1018.195,297.313,-139.036,169.953,50.705,159.810
C06969=1018.201,297.561,-139.068,169.958,50.700,159.810
C06970=1018.207,297.809,-139.099,169.964,50.696,159.810
C06971=1018.213,298.057,-139.131,169.970,50.692,159.810
C06972=1018.220,298.304,-139.163,169.976,50.687,159.810
C06973=1018.226,298.552,-139.195,169.981,50.683,159.810
C06974=1018.233,298.800,-139.226,169.987,50.679,159.810
C06975=1018.239,299.048,-139.258,169.993,50.674,159.810
C06976=1018.245,299.296,-139.289,169.997,50.670,159.810
C06977=1018.251,299.544,-139.321,170.003,50.666,159.810
C06978=1018.257,299.791,-139.354,170.009,50.662,159.810
C06979=1018.264,300.039,-139.386,170.014,50.658,159.810
C06980=1018.270,300.288,-139.418,170.020,50.653,159.810
C06981=1018.277,300.535,-139.450,170.026,50.649,159.810
C06982=1018.283,300.783,-139.482,170.032,50.644,159.810
C06983=1018.290,301.031,-139.513,170.037,50.641,159.810
C06984=1018.296,301.279,-139.545,170.043,50.637,159.810
C06985=1018.303,301.527,-139.577,170.048,50.632,159.810
C06986=1018.308,301.774,-139.609,170.053,50.628,159.810
C06987=1018.314,302.022,-139.641,170.059,50.624,159.810
C06988=1018.321,302.270,-139.673,170.065,50.620,159.810
C06989=1018.327,302.518,-139.705,170.071,50.616,159.810
C06990=1018.334,302.765,-139.737,170.076,50.612,159.810
C06991=1018.340,303.013,-139.770,170.082,50.607,159.810
C06992=1018.347,303.260,-139.802,170.088,50.603,159.810
C06993=1018.353,303.509,-139.834,170.094,50.599,159.810
C06994=1018.360,303.756,-139.866,170.099,50.595,159.810
C06995=1018.367,304.005,-139.898,170.105,50.591,159.810
C06996=1018.373,304.253,-139.931,170.111,50.586,159.810
C06997=1018.380,304.500,-139.962,170.117,50.583,159.810
C06998=1018.386,304.748,-139.995,170.122,50.579,159.810
C06999=1018.393,304.996,-140.027,170.128,50.574,159.810
C07000=1018.399,305.243,-140.059,170.134,50.571,159.811
C07001=1018.405,305.492,-140.091,170.139,50.567,159.810
C07002=1018.412,305.739,-140.123,170.145,50.562,159.810
C07003=1018.419,305.987,-140.156,170.151,50.559,159.811
C07004=1018.425,306.234,-140.188,170.157,50.554,159.811
C07005=1018.432,306.482,-140.220,170.163,50.550,159.811
C07006=1018.439,306.730,-140.253,170.168,50.546,159.811
C07007=1018.445,306.978,-140.285,170.174,50.543,159.811
C07008=1018.451,307.226,-140.318,170.180,50.538,159.811
C07009=1018.459,307.474,-140.349,170.186,50.534,159.811
C07010=1018.465,307.722,-140.382,170.191,50.531,159.811
C07011=1018.472,307.971,-140.415,170.197,50.526,159.811
C07012=1018.479,308.218,-140.447,170.203,50.522,159.811
C07013=1018.485,308.466,-140.480,170.210,50.519,159.812
C07014=1018.491,308.713,-140.512,170.214,50.515,159.811
C07015=1018.499,308.961,-140.545,170.221,50.511,159.812
C07016=1018.505,309.209,-140.578,170.227,50.507,159.812
C07017=1018.512,309.456,-140.610,170.233,50.503,159.812
C07018=1018.518,309.705,-140.642,170.239,50.499,159.812
C07019=1018.525,309.951,-140.675,170.244,50.495,159.812
C07020=1018.532,310.200,-140.708,170.250,50.492,159.812
C07021=1018.538,310.447,-140.741,170.256,50.488,159.812
C07022=1018.544,310.695,-140.774,170.262,50.484,159.812
C07023=1018.550,310.943,-140.807,170.268,50.481,159.813
C07024=1018.557,311.191,-140.841,170.274,50.477,159.813
C07025=1018.563,311.438,-140.874,170.279,50.474,159.813
C07026=1018.570,311.686,-140.906,170.285,50.469,159.813
C07027=1018.575,311.933,-140.940,170.292,50.466,159.813
C07028=1018.582,312.181,-140.974,170.297,50.462,159.813
C07029=1018.589,312.429,-141.006,170.303,50.458,159.813
C07030=1018.595,312.676,-141.040,170.309,50.455,159.814
C07031=1018.602,312.924,-141.073,170.315,50.451,159.814
C07032=1018.608,313.172,-141.106,170.321,50.448,159.814
C07033=1018.614,313.419,-141.140,170.327,50.444,159.814
C07034=1018.621,313.667,-141.173,170.333,50.440,159.814
C07035=1018.628,313.914,-141.206,170.339,50.438,159.815
C07036=1018.633,314.162,-141.240,170.345,50.434,159.815
C07037=1018.641,314.410,-141.273,170.351,50.430,159.815
C07038=1018.647,314.657,-141.306,170.357,50.427,159.815
C07039=1018.654,314.905,-141.340,170.363,50.423,159.815
C07040=1018.660,315.153,-141.373,170.369,50.419,159.816
C07041=1018.666,315.400,-141.407,170.374,50.416,159.816
C07042=1018.673,315.648,-141.440,170.381,50.412,159.816
C07043=1018.680,315.895,-141.473,170.387,50.409,159.816
C07044=1018.687,316.144,-141.506,170.394,50.406,159.817
C07045=1018.692,316.391,-141.540,170.399,50.402,159.817
C07046=1018.700,316.639,-141.574,170.405,50.399,159.817
C07047=1018.706,316.886,-141.607,170.411,50.395,159.817
C07048=1018.713,317.134,-141.641,170.418,50.392,159.817
C07049=1018.719,317.381,-141.675,170.423,50.388,159.818
C07050=1018.726,317.629,-141.708,170.430,50.385,159.818
C07051=1018.733,317.877,-141.742,170.436,50.382,159.818
C07052=1018.740,318.124,-141.775,170.442,50.378,159.818
C07053=1018.746,318.373,-141.809,170.448,50.375,159.818
C07054=1018.752,318.620,-141.842,170.454,50.371,159.819
C07055=1018.760,318.867,-141.876,170.461,50.368,159.819
C07056=1018.767,319.115,-141.910,170.467,50.364,159.819
C07057=1018.773,319.362,-141.944,170.473,50.361,159.820
C07058=1018.780,319.611,-141.977,170.479,50.358,159.820
C07059=1018.786,319.858,-142.011,170.485,50.354,159.820
C07060=1018.793,320.105,-142.045,170.492,50.351,159.820
C07061=1018.800,320.353,-142.079,170.498,50.347,159.821
C07062=1018.807,320.601,-142.113,170.504,50.345,159.821
C07063=1018.814,320.848,-142.146,170.510,50.341,159.821
C07064=1018.821,321.096,-142.180,170.516,50.338,159.821
C07065=1018.827,321.344,-142.215,170.523,50.334,159.822
C07066=1018.834,321.590,-142.248,170.529,50.331,159.822
C07067=1018.841,321.838,-142.282,170.535,50.328,159.822
C07068=1018.848,322.092,-142.317,170.541,50.325,159.823
C07069=1018.855,322.345,-142.351,170.548,50.321,159.823
C07070=1018.863,322.598,-142.386,170.554,50.318,159.823
C07071=1018.870,322.852,-142.421,170.560,50.314,159.823
C07072=1018.877,323.100,-142.455,170.567,50.311,159.824
C07073=1018.883,323.347,-142.488,170.574,50.308,159.824
C07074=1018.890,323.595,-142.523,170.580,50.305,159.824
C07075=1018.897,323.843,-142.557,170.587,50.301,159.825
C07076=1018.904,324.090,-142.590,170.592,50.299,159.825
C07077=1018.911,324.338,-142.625,170.598,50.295,159.825
C07078=1018.918,324.586,-142.659,170.605,50.292,159.826
C07079=1018.925,324.833,-142.693,170.612,50.289,159.826
C07080=1018.933,325.081,-142.727,170.618,50.286,159.826
C07081=1018.939,325.328,-142.761,170.625,50.282,159.827
C07082=1018.946,325.576,-142.795,170.630,50.280,159.827
C07083=1018.953,325.823,-142.829,170.637,50.277,159.827
C07084=1018.960,326.070,-142.863,170.644,50.273,159.828
C07085=1018.967,326.318,-142.898,170.650,50.270,159.828
C07086=1018.974,326.565,-142.932,170.656,50.267,159.828
C07087=1018.981,326.813,-142.967,170.663,50.264,159.829
C07088=1018.988,327.061,-143.002,170.669,50.261,159.829
C07089=1018.995,327.308,-143.036,170.675,50.258,159.829
C07090=1019.002,327.556,-143.071,170.682,50.256,159.830
C07091=1019.008,327.803,-143.106,170.689,50.253,159.830
C07092=1019.016,328.051,-143.140,170.696,50.249,159.831
C07093=1019.022,328.298,-143.175,170.701,50.247,159.831
C07094=1019.029,328.546,-143.210,170.708,50.244,159.831
C07095=1019.036,328.793,-143.244,170.715,50.241,159.832
C07096=1019.043,329.041,-143.279,170.721,50.238,159.832
C07097=1019.050,329.288,-143.314,170.728,50.235,159.833
C07098=1019.057,329.535,-143.349,170.735,50.232,159.833
C07099=1019.064,329.783,-143.383,170.741,50.230,159.834
C07100=1019.071,330.030,-143.418,170.747,50.226,159.834
C07101=1019.077,330.278,-143.453,170.754,50.223,159.834
C07102=1019.085,330.526,-143.488,170.760,50.220,159.835
C07103=1019.092,330.773,-143.523,170.767,50.217,159.835
C07104=1019.099,331.021,-143.558,170.774,50.215,159.836
C07105=1019.105,331.268,-143.593,170.780,50.212,159.836
C07106=1019.113,331.515,-143.627,170.786,50.209,159.836
C07107=1019.120,331.763,-143.663,170.793,50.207,159.837
C07108=1019.127,332.011,-143.698,170.800,50.204,159.837
C07109=1019.134,332.258,-143.733,170.807,50.201,159.838
C07110=1019.141,332.505,-143.768,170.814,50.198,159.838
C07111=1019.148,332.752,-143.803,170.820,50.195,159.839
C07112=1019.155,333.000,-143.838,170.827,50.193,159.839
C07113=1019.162,333.248,-143.874,170.833,50.190,159.840
C07114=1019.169,333.495,-143.909,170.840,50.188,159.840
C07115=1019.176,333.742,-143.945,170.847,50.185,159.841
C07116=1019.183,333.989,-143.980,170.854,50.182,159.841
C07117=1019.190,334.237,-144.015,170.860,50.179,159.842
C07118=1019.197,334.485,-144.050,170.867,50.177,159.842
C07119=1019.204,334.732,-144.086,170.874,50.174,159.843
C07120=1019.211,334.979,-144.121,170.880,50.172,159.843
C07121=1019.218,335.227,-144.157,170.887,50.169,159.844
C07122=1019.225,335.474,-144.193,170.894,50.166,159.844
C07123=1019.232,335.721,-144.228,170.901,50.164,159.845
C07124=1019.239,335.969,-144.263,170.908,50.162,159.845
C07125=1019.247,336.216,-144.299,170.914,50.159,159.846
C07126=1019.253,336.463,-144.334,170.921,50.156,159.846
C07127=1019.261,336.711,-144.370,170.928,50.154,159.847
C07128=1019.269,336.960,-144.406,170.935,50.151,159.847
C07129=1019.276,337.209,-144.442,170.942,50.148,159.848
C07130=1019.283,337.459,-144.478,170.949,50.146,159.848
C07131=1019.290,337.707,-144.513,170.956,50.144,159.849
C07132=1019.298,337.955,-144.549,170.963,50.141,159.849
C07133=1019.305,338.202,-144.585,170.970,50.138,159.850
C07134=1019.312,338.450,-144.620,170.976,50.136,159.851
C07135=1019.319,338.697,-144.656,170.983,50.134,159.851
C07136=1019.327,338.944,-144.692,170.990,50.131,159.852
C07137=1019.333,339.191,-144.727,170.997,50.129,159.852
C07138=1019.340,339.439,-144.764,171.004,50.126,159.853
C07139=1019.347,339.686,-144.800,171.011,50.124,159.854
C07140=1019.355,339.933,-144.836,171.018,50.122,159.854
C07141=1019.362,340.181,-144.871,171.025,50.119,159.855
C07142=1019.370,340.428,-144.908,171.032,50.117,159.855
C07143=1019.377,340.676,-144.944,171.039,50.115,159.856
C07144=1019.384,340.923,-144.980,171.046,50.112,159.856
C07145=1019.391,341.170,-145.016,171.053,50.110,159.857
C07146=1019.398,341.417,-145.052,171.060,50.107,159.858
C07147=1019.405,341.665,-145.089,171.067,50.105,159.858
C07148=1019.413,341.912,-145.125,171.074,50.103,159.859
C07149=1019.420,342.159,-145.161,171.082,50.101,159.860
C07150=1019.428,342.406,-145.197,171.089,50.098,159.860
C07151=1019.435,342.654,-145.234,171.096,50.096,159.861
C07152=1019.442,342.901,-145.270,171.103,50.094,159.862
C07153=1019.449,343.148,-145.306,171.110,50.092,159.862
C07154=1019.457,343.396,-145.343,171.117,50.089,159.863
C07155=1019.463,343.643,-145.379,171.124,50.087,159.863
C07156=1019.471,343.890,-145.415,171.131,50.085,159.864
C07157=1019.479,344.137,-145.452,171.138,50.083,159.865
C07158=1019.486,344.385,-145.489,171.145,50.080,159.865
C07159=1019.493,344.632,-145.525,171.153,50.079,159.866
C07160=1019.501,344.879,-145.561,171.160,50.076,159.867
